LIN {X 0,Y 522.587,Z 549.53,A -85,B 0,C 180,E1 4793.93,E2 4793.93} C_VEL
LIN {X 0,Y 522.386,Z 549.53,A -85,B 0,C 180,E1 4799.594,E2 4799.594} C_VEL
LIN {X 0,Y 522.323,Z 549.53,A -85,B 0,C 180,E1 4805.74,E2 4805.74} C_VEL
LIN {X 0,Y 522.361,Z 549.53,A -85,B 0,C 180,E1 4811.419,E2 4811.419} C_VEL
LIN {X 0,Y 533.947,Z 582.684,A -85,B 0,C 180,E1 4813.515,E2 4813.515} C_VEL
LIN {X 0,Y 531.782,Z 621.229,A -85,B 0,C 180,E1 4815.534,E2 4815.534} C_VEL
LIN {X 0,Y 529.396,Z 657.061,A -85,B 0,C 180,E1 4818.174,E2 4818.174} C_VEL
LIN {X 0,Y 527.169,Z 689.396,A -85,B 0,C 180,E1 4821.377,E2 4821.377} C_VEL
LIN {X 0,Y 525.44,Z 717.104,A -85,B 0,C 180,E1 4824.999,E2 4824.999} C_VEL
LIN {X 0,Y 524.207,Z 740.402,A -85,B 0,C 180,E1 4829.059,E2 4829.059} C_VEL
LIN {X 0,Y 523.575,Z 757.4,A -85,B 0,C 180,E1 4833.13,E2 4833.13} C_VEL
LIN {X 0,Y 523.223,Z 768.491,A -85,B 0,C 180,E1 4837.003,E2 4837.003} C_VEL
LIN {X 0,Y 522.979,Z 775.702,A -85,B 0,C 180,E1 4841.427,E2 4841.427} C_VEL
LIN {X 0,Y 523.022,Z 777.495,A -85,B 0,C 180,E1 4844.895,E2 4844.895} C_VEL
LIN {X 0,Y 523.078,Z 775.878,A -85,B 0,C 180,E1 4848.307,E2 4848.307} C_VEL
LIN {X 0,Y 523.253,Z 769.377,A -85,B 0,C 180,E1 4852.515,E2 4852.515} C_VEL
LIN {X 0,Y 523.557,Z 757.742,A -85,B 0,C 180,E1 4856.681,E2 4856.681} C_VEL
LIN {X 0,Y 524.184,Z 739.509,A -85,B 0,C 180,E1 4861.031,E2 4861.031} C_VEL
LIN {X 0,Y 525.342,Z 716.823,A -85,B 0,C 180,E1 4864.956,E2 4864.956} C_VEL
LIN {X 0,Y 527.118,Z 690.017,A -85,B 0,C 180,E1 4868.461,E2 4868.461} C_VEL
LIN {X 0,Y 529.345,Z 658.044,A -85,B 0,C 180,E1 4871.65,E2 4871.65} C_VEL
LIN {X 0,Y 531.728,Z 622.755,A -85,B 0,C 180,E1 4874.276,E2 4874.276} C_VEL
LIN {X 0,Y 533.842,Z 585.818,A -85,B 0,C 180,E1 4876.253,E2 4876.253} C_VEL
LIN {X 0,Y 533.35,Z 577.741,A -85,B 0,C 180,E1 4876.653,E2 4876.653} C_VEL
LIN {X 0,Y 522.59,Z 549.53,A -85,B 0,C 180,E1 4878.475,E2 4878.475} C_VEL
LIN {X 0,Y 522.511,Z 549.53,A -85,B 0,C 180,E1 4879.609,E2 4879.609} C_VEL
LIN {X 0,Y 520.002,Z 549.53,A -85,B 0,C 180,E1 4881.019,E2 4881.019} C_VEL
LIN {X 0,Y 514.659,Z 549.53,A -85,B 0,C 180,E1 4883.132,E2 4883.132} C_VEL
LIN {X 0,Y 514.565,Z 549.53,A -85,B 0,C 180,E1 4883.376,E2 4883.376} C_VEL
LIN {X 0,Y 514.494,Z 549.53,A -85,B 0,C 180,E1 4888.085,E2 4888.085} C_VEL
LIN {X 0,Y 514.37,Z 549.53,A -85,B 0,C 180,E1 4894,E2 4894} C_VEL
LIN {X 0,Y 514.463,Z 549.53,A -85,B 0,C 180,E1 4900.344,E2 4900.344} C_VEL
LIN {X 0,Y 514.4,Z 549.53,A -85,B 0,C 180,E1 4905.056,E2 4905.056} C_VEL
LIN {X 0,Y 514.337,Z 549.53,A -85,B 0,C 180,E1 4911.816,E2 4911.816} C_VEL
LIN {X 0,Y 514.446,Z 549.53,A -85,B 0,C 180,E1 4914.365,E2 4914.365} C_VEL
LIN {X 0,Y 529.549,Z 582.461,A -85,B 0,C 180,E1 4916.004,E2 4916.004} C_VEL
LIN {X 0,Y 528.701,Z 628.433,A -85,B 0,C 180,E1 4916.908,E2 4916.908} C_VEL
LIN {X 0,Y 526.969,Z 666.113,A -85,B 0,C 180,E1 4918.265,E2 4918.265} C_VEL
LIN {X 0,Y 524.654,Z 702.724,A -85,B 0,C 180,E1 4920.246,E2 4920.246} C_VEL
LIN {X 0,Y 522.113,Z 737.095,A -85,B 0,C 180,E1 4922.823,E2 4922.823} C_VEL
LIN {X 0,Y 519.796,Z 768.223,A -85,B 0,C 180,E1 4925.933,E2 4925.933} C_VEL
LIN {X 0,Y 517.817,Z 795.232,A -85,B 0,C 180,E1 4929.459,E2 4929.459} C_VEL
LIN {X 0,Y 516.475,Z 818.065,A -85,B 0,C 180,E1 4933.391,E2 4933.391} C_VEL
LIN {X 0,Y 515.7,Z 834.826,A -85,B 0,C 180,E1 4937.279,E2 4937.279} C_VEL
LIN {X 0,Y 515.364,Z 847.612,A -85,B 0,C 180,E1 4941.552,E2 4941.552} C_VEL
LIN {X 0,Y 515.231,Z 853.932,A -85,B 0,C 180,E1 4944.942,E2 4944.942} C_VEL
LIN {X 0,Y 515.211,Z 857.084,A -85,B 0,C 180,E1 4948.315,E2 4948.315} C_VEL
LIN {X 0,Y 515.199,Z 856.636,A -85,B 0,C 180,E1 4952.428,E2 4952.428} C_VEL
LIN {X 0,Y 515.289,Z 851.182,A -85,B 0,C 180,E1 4956.749,E2 4956.749} C_VEL
LIN {X 0,Y 515.5,Z 841.923,A -85,B 0,C 180,E1 4960.589,E2 4960.589} C_VEL
LIN {X 0,Y 516.106,Z 826.652,A -85,B 0,C 180,E1 4964.776,E2 4964.776} C_VEL
LIN {X 0,Y 517.278,Z 804.95,A -85,B 0,C 180,E1 4969.003,E2 4969.003} C_VEL
LIN {X 0,Y 519.005,Z 778.608,A -85,B 0,C 180,E1 4972.821,E2 4972.821} C_VEL
LIN {X 0,Y 521.271,Z 748.093,A -85,B 0,C 180,E1 4976.175,E2 4976.175} C_VEL
LIN {X 0,Y 523.839,Z 713.836,A -85,B 0,C 180,E1 4979.007,E2 4979.007} C_VEL
LIN {X 0,Y 526.461,Z 675.681,A -85,B 0,C 180,E1 4981.288,E2 4981.288} C_VEL
LIN {X 0,Y 528.473,Z 635.637,A -85,B 0,C 180,E1 4982.884,E2 4982.884} C_VEL
LIN {X 0,Y 529.548,Z 593.899,A -85,B 0,C 180,E1 4983.813,E2 4983.813} C_VEL
LIN {X 0,Y 528.896,Z 580.557,A -85,B 0,C 180,E1 4984.075,E2 4984.075} C_VEL
LIN {X 0,Y 514.406,Z 549.53,A -85,B 0,C 180,E1 4985.73,E2 4985.73} C_VEL
LIN {X 0,Y 514.463,Z 549.53,A -85,B 0,C 180,E1 4990.349,E2 4990.349} C_VEL
LIN {X 0,Y 514.395,Z 549.53,A -85,B 0,C 180,E1 4995.063,E2 4995.063} C_VEL
LIN {X 0,Y 514.324,Z 549.53,A -85,B 0,C 180,E1 5001.821,E2 5001.821} C_VEL
LIN {X 0,Y 514.526,Z 549.53,A -85,B 0,C 180,E1 5008.022,E2 5008.022} C_VEL
LIN {X 0,Y 514.498,Z 549.53,A -85,B 0,C 180,E1 5013.81,E2 5013.81} C_VEL
LIN {X 0,Y 514.563,Z 549.53,A -85,B 0,C 180,E1 5019.328,E2 5019.328} C_VEL
LIN {X 0,Y 514.73,Z 549.53,A -85,B 0,C 180,E1 5024.653,E2 5024.653} C_VEL
LIN {X 0,Y 514.859,Z 549.53,A -85,B 0,C 180,E1 5029.841,E2 5029.841} C_VEL
LIN {X 0,Y 514.93,Z 549.53,A -85,B 0,C 180,E1 5034.943,E2 5034.943} C_VEL
LIN {X 0,Y 515.174,Z 549.53,A -85,B 0,C 180,E1 5041.688,E2 5041.688} C_VEL
LIN {X 0,Y 515.005,Z 549.53,A -85,B 0,C 180,E1 5046.757,E2 5046.757} C_VEL
LIN {X 0,Y 514.781,Z 549.53,A -85,B 0,C 180,E1 5051.884,E2 5051.884} C_VEL
LIN {X 0,Y 514.696,Z 549.53,A -85,B 0,C 180,E1 5057.111,E2 5057.111} C_VEL
LIN {X 0,Y 514.62,Z 549.53,A -85,B 0,C 180,E1 5062.49,E2 5062.49} C_VEL
LIN {X 0,Y 514.462,Z 549.53,A -85,B 0,C 180,E1 5068.095,E2 5068.095} C_VEL
LIN {X 0,Y 514.358,Z 549.53,A -85,B 0,C 180,E1 5074.01,E2 5074.01} C_VEL
LIN {X 0,Y 514.423,Z 549.53,A -85,B 0,C 180,E1 5080.358,E2 5080.358} C_VEL
LIN {X 0,Y 514.362,Z 549.53,A -85,B 0,C 180,E1 5085.054,E2 5085.054} C_VEL
LIN {X 0,Y 514.345,Z 549.53,A -85,B 0,C 180,E1 5089.942,E2 5089.942} C_VEL
LIN {X 0,Y 514.429,Z 549.53,A -85,B 0,C 180,E1 5096,E2 5096} C_VEL
LIN {X 0,Y 514.46,Z 549.53,A -85,B 0,C 180,E1 5101.999,E2 5101.999} C_VEL
LIN {X 0,Y 514.558,Z 549.53,A -85,B 0,C 180,E1 5107.511,E2 5107.511} C_VEL
LIN {X 0,Y 514.696,Z 549.53,A -85,B 0,C 180,E1 5112.893,E2 5112.893} C_VEL
LIN {X 0,Y 514.781,Z 549.53,A -85,B 0,C 180,E1 5118.12,E2 5118.12} C_VEL
LIN {X 0,Y 514.881,Z 549.53,A -85,B 0,C 180,E1 5123.246,E2 5123.246} C_VEL
LIN {X 0,Y 514.971,Z 549.53,A -85,B 0,C 180,E1 5128.524,E2 5128.524} C_VEL
LIN {X 0,Y 514.933,Z 549.53,A -85,B 0,C 180,E1 5133.372,E2 5133.372} C_VEL
LIN {X 0,Y 514.812,Z 549.53,A -85,B 0,C 180,E1 5138.457,E2 5138.457} C_VEL
LIN {X 0,Y 514.743,Z 549.53,A -85,B 0,C 180,E1 5143.904,E2 5143.904} C_VEL
LIN {X 0,Y 514.64,Z 549.53,A -85,B 0,C 180,E1 5149.7,E2 5149.7} C_VEL
LIN {X 0,Y 514.658,Z 549.53,A -85,B 0,C 180,E1 5154.323,E2 5154.323} C_VEL
LIN {X 0,Y 514.447,Z 549.53,A -85,B 0,C 180,E1 5160.022,E2 5160.022} C_VEL
LIN {X 0,Y 514.412,Z 549.53,A -85,B 0,C 180,E1 5166.063,E2 5166.063} C_VEL
LIN {X 0,Y 514.465,Z 550.037,A -85,B 0,C 180,E1 5170.866,E2 5170.866} C_VEL
LIN {X 0,Y 527.106,Z 583.478,A -85,B 0,C 180,E1 5173.098,E2 5173.098} C_VEL
LIN {X 0,Y 524.76,Z 621.631,A -85,B 0,C 180,E1 5175.128,E2 5175.128} C_VEL
LIN {X 0,Y 522.259,Z 655.644,A -85,B 0,C 180,E1 5177.647,E2 5177.647} C_VEL
LIN {X 0,Y 519.773,Z 688.501,A -85,B 0,C 180,E1 5180.915,E2 5180.915} C_VEL
LIN {X 0,Y 517.796,Z 716.835,A -85,B 0,C 180,E1 5184.65,E2 5184.65} C_VEL
LIN {X 0,Y 516.485,Z 739.169,A -85,B 0,C 180,E1 5188.564,E2 5188.564} C_VEL
LIN {X 0,Y 515.708,Z 757.505,A -85,B 0,C 180,E1 5192.977,E2 5192.977} C_VEL
LIN {X 0,Y 515.274,Z 769.934,A -85,B 0,C 180,E1 5197.54,E2 5197.54} C_VEL
LIN {X 0,Y 515.086,Z 775.461,A -85,B 0,C 180,E1 5201.132,E2 5201.132} C_VEL
LIN {X 0,Y 515.088,Z 777.462,A -85,B 0,C 180,E1 5204.657,E2 5204.657} C_VEL
LIN {X 0,Y 515.153,Z 776.109,A -85,B 0,C 180,E1 5208.124,E2 5208.124} C_VEL
LIN {X 0,Y 515.348,Z 769.867,A -85,B 0,C 180,E1 5212.399,E2 5212.399} C_VEL
LIN {X 0,Y 515.68,Z 758.507,A -85,B 0,C 180,E1 5216.63,E2 5216.63} C_VEL
LIN {X 0,Y 516.358,Z 740.653,A -85,B 0,C 180,E1 5221.047,E2 5221.047} C_VEL
LIN {X 0,Y 517.728,Z 716.827,A -85,B 0,C 180,E1 5225.263,E2 5225.263} C_VEL
LIN {X 0,Y 519.792,Z 688.415,A -85,B 0,C 180,E1 5229.004,E2 5229.004} C_VEL
LIN {X 0,Y 522.267,Z 655.937,A -85,B 0,C 180,E1 5232.235,E2 5232.235} C_VEL
LIN {X 0,Y 524.895,Z 620.24,A -85,B 0,C 180,E1 5234.87,E2 5234.87} C_VEL
LIN {X 0,Y 527.04,Z 581.921,A -85,B 0,C 180,E1 5236.891,E2 5236.891} C_VEL
LIN {X 0,Y 514.633,Z 549.53,A -85,B 0,C 180,E1 5239.082,E2 5239.082} C_VEL
LIN {X 0,Y 514.565,Z 549.53,A -85,B 0,C 180,E1 5243.376,E2 5243.376} C_VEL
LIN {X 0,Y 512.046,Z 549.53,A -85,B 0,C 180,E1 5244.81,E2 5244.81} C_VEL
LIN {X 0,Y 506.53,Z 549.53,A -85,B 0,C 180,E1 5247.208,E2 5247.208} C_VEL
LIN {X 0,Y 506.407,Z 549.53,A -85,B 0,C 180,E1 5253.158,E2 5253.158} C_VEL
LIN {X 0,Y 506.467,Z 549.53,A -85,B 0,C 180,E1 5258.988,E2 5258.988} C_VEL
LIN {X 0,Y 506.44,Z 549.53,A -85,B 0,C 180,E1 5264.15,E2 5264.15} C_VEL
LIN {X 0,Y 506.376,Z 549.53,A -85,B 0,C 180,E1 5268.867,E2 5268.867} C_VEL
LIN {X 0,Y 506.525,Z 549.563,A -85,B 0,C 180,E1 5273.887,E2 5273.887} C_VEL
LIN {X 0,Y 514.606,Z 567.373,A -85,B 0,C 180,E1 5274.676,E2 5274.676} C_VEL
LIN {X 0,Y 522.982,Z 584.842,A -85,B 0,C 180,E1 5275.556,E2 5275.556} C_VEL
LIN {X 0,Y 522.081,Z 628.432,A -85,B 0,C 180,E1 5276.433,E2 5276.433} C_VEL
LIN {X 0,Y 520.149,Z 666.955,A -85,B 0,C 180,E1 5277.842,E2 5277.842} C_VEL
LIN {X 0,Y 517.68,Z 702.721,A -85,B 0,C 180,E1 5279.804,E2 5279.804} C_VEL
LIN {X 0,Y 514.937,Z 737.092,A -85,B 0,C 180,E1 5282.412,E2 5282.412} C_VEL
LIN {X 0,Y 512.366,Z 768.222,A -85,B 0,C 180,E1 5285.561,E2 5285.561} C_VEL
LIN {X 0,Y 510.225,Z 795.231,A -85,B 0,C 180,E1 5289.139,E2 5289.139} C_VEL
LIN {X 0,Y 508.729,Z 818.063,A -85,B 0,C 180,E1 5293.131,E2 5293.131} C_VEL
LIN {X 0,Y 507.884,Z 834.827,A -85,B 0,C 180,E1 5297.08,E2 5297.08} C_VEL
LIN {X 0,Y 507.481,Z 847.612,A -85,B 0,C 180,E1 5301.42,E2 5301.42} C_VEL
LIN {X 0,Y 507.334,Z 853.932,A -85,B 0,C 180,E1 5304.863,E2 5304.863} C_VEL
LIN {X 0,Y 507.329,Z 857.084,A -85,B 0,C 180,E1 5308.289,E2 5308.289} C_VEL
LIN {X 0,Y 507.391,Z 857.086,A -85,B 0,C 180,E1 5311.709,E2 5311.709} C_VEL
LIN {X 0,Y 507.418,Z 852.726,A -85,B 0,C 180,E1 5315.994,E2 5315.994} C_VEL
LIN {X 0,Y 507.617,Z 843.214,A -85,B 0,C 180,E1 5320.309,E2 5320.309} C_VEL
LIN {X 0,Y 508.243,Z 827.853,A -85,B 0,C 180,E1 5324.727,E2 5324.727} C_VEL
LIN {X 0,Y 509.531,Z 806.274,A -85,B 0,C 180,E1 5329.078,E2 5329.078} C_VEL
LIN {X 0,Y 511.324,Z 781.087,A -85,B 0,C 180,E1 5332.858,E2 5332.858} C_VEL
LIN {X 0,Y 513.741,Z 751.547,A -85,B 0,C 180,E1 5336.235,E2 5336.235} C_VEL
LIN {X 0,Y 516.505,Z 717.528,A -85,B 0,C 180,E1 5339.169,E2 5339.169} C_VEL
LIN {X 0,Y 519.259,Z 681.482,A -85,B 0,C 180,E1 5341.44,E2 5341.44} C_VEL
LIN {X 0,Y 521.439,Z 645.004,A -85,B 0,C 180,E1 5343.038,E2 5343.038} C_VEL
LIN {X 0,Y 522.843,Z 606.759,A -85,B 0,C 180,E1 5344.069,E2 5344.069} C_VEL
LIN {X 0,Y 522.345,Z 583.286,A -85,B 0,C 180,E1 5344.517,E2 5344.517} C_VEL
LIN {X 0,Y 506.501,Z 549.53,A -85,B 0,C 180,E1 5346.278,E2 5346.278} C_VEL
LIN {X 0,Y 506.498,Z 549.53,A -85,B 0,C 180,E1 5351.648,E2 5351.648} C_VEL
LIN {X 0,Y 506.4,Z 549.53,A -85,B 0,C 180,E1 5356.561,E2 5356.561} C_VEL
LIN {X 0,Y 506.445,Z 549.53,A -85,B 0,C 180,E1 5363.285,E2 5363.285} C_VEL
LIN {X 0,Y 506.581,Z 549.53,A -85,B 0,C 180,E1 5369.468,E2 5369.468} C_VEL
LIN {X 0,Y 506.579,Z 549.53,A -85,B 0,C 180,E1 5375.269,E2 5375.269} C_VEL
LIN {X 0,Y 506.698,Z 549.53,A -85,B 0,C 180,E1 5380.815,E2 5380.815} C_VEL
LIN {X 0,Y 506.872,Z 549.53,A -85,B 0,C 180,E1 5386.179,E2 5386.179} C_VEL
LIN {X 0,Y 506.99,Z 549.53,A -85,B 0,C 180,E1 5391.416,E2 5391.416} C_VEL
LIN {X 0,Y 507.148,Z 549.53,A -85,B 0,C 180,E1 5396.581,E2 5396.581} C_VEL
LIN {X 0,Y 507.283,Z 549.53,A -85,B 0,C 180,E1 5401.714,E2 5401.714} C_VEL
LIN {X 0,Y 507.076,Z 549.53,A -85,B 0,C 180,E1 5406.863,E2 5406.863} C_VEL
LIN {X 0,Y 506.851,Z 549.53,A -85,B 0,C 180,E1 5412.073,E2 5412.073} C_VEL
LIN {X 0,Y 506.779,Z 549.53,A -85,B 0,C 180,E1 5417.387,E2 5417.387} C_VEL
LIN {X 0,Y 506.704,Z 549.53,A -85,B 0,C 180,E1 5422.861,E2 5422.861} C_VEL
LIN {X 0,Y 506.497,Z 549.53,A -85,B 0,C 180,E1 5428.577,E2 5428.577} C_VEL
LIN {X 0,Y 506.449,Z 549.53,A -85,B 0,C 180,E1 5434.615,E2 5434.615} C_VEL
LIN {X 0,Y 506.433,Z 549.53,A -85,B 0,C 180,E1 5441.13,E2 5441.13} C_VEL
LIN {X 0,Y 506.356,Z 549.53,A -85,B 0,C 180,E1 5446.551,E2 5446.551} C_VEL
LIN {X 0,Y 506.448,Z 549.53,A -85,B 0,C 180,E1 5453.28,E2 5453.28} C_VEL
LIN {X 0,Y 506.573,Z 549.53,A -85,B 0,C 180,E1 5459.463,E2 5459.463} C_VEL
LIN {X 0,Y 506.586,Z 549.53,A -85,B 0,C 180,E1 5465.266,E2 5465.266} C_VEL
LIN {X 0,Y 506.732,Z 549.53,A -85,B 0,C 180,E1 5470.813,E2 5470.813} C_VEL
LIN {X 0,Y 506.888,Z 549.53,A -85,B 0,C 180,E1 5476.176,E2 5476.176} C_VEL
LIN {X 0,Y 506.985,Z 549.53,A -85,B 0,C 180,E1 5481.413,E2 5481.413} C_VEL
LIN {X 0,Y 507.204,Z 549.53,A -85,B 0,C 180,E1 5486.578,E2 5486.578} C_VEL
LIN {X 0,Y 507.286,Z 549.53,A -85,B 0,C 180,E1 5491.711,E2 5491.711} C_VEL
LIN {X 0,Y 507.096,Z 549.53,A -85,B 0,C 180,E1 5496.86,E2 5496.86} C_VEL
LIN {X 0,Y 506.879,Z 549.53,A -85,B 0,C 180,E1 5502.07,E2 5502.07} C_VEL
LIN {X 0,Y 506.801,Z 549.53,A -85,B 0,C 180,E1 5507.383,E2 5507.383} C_VEL
LIN {X 0,Y 506.747,Z 549.53,A -85,B 0,C 180,E1 5512.857,E2 5512.857} C_VEL
LIN {X 0,Y 506.55,Z 549.53,A -85,B 0,C 180,E1 5518.571,E2 5518.571} C_VEL
LIN {X 0,Y 506.478,Z 549.53,A -85,B 0,C 180,E1 5524.611,E2 5524.611} C_VEL
LIN {X 0,Y 506.565,Z 549.913,A -85,B 0,C 180,E1 5530.288,E2 5530.288} C_VEL
LIN {X 0,Y 520.194,Z 586.345,A -85,B 0,C 180,E1 5532.764,E2 5532.764} C_VEL
LIN {X 0,Y 517.628,Z 624.022,A -85,B 0,C 180,E1 5534.842,E2 5534.842} C_VEL
LIN {X 0,Y 514.887,Z 657.943,A -85,B 0,C 180,E1 5537.439,E2 5537.439} C_VEL
LIN {X 0,Y 512.251,Z 689.781,A -85,B 0,C 180,E1 5540.693,E2 5540.693} C_VEL
LIN {X 0,Y 510.115,Z 717.806,A -85,B 0,C 180,E1 5544.485,E2 5544.485} C_VEL
LIN {X 0,Y 508.63,Z 740.964,A -85,B 0,C 180,E1 5548.676,E2 5548.676} C_VEL
LIN {X 0,Y 507.84,Z 758.04,A -85,B 0,C 180,E1 5552.954,E2 5552.954} C_VEL
LIN {X 0,Y 507.438,Z 769.407,A -85,B 0,C 180,E1 5557.174,E2 5557.174} C_VEL
LIN {X 0,Y 507.203,Z 775.22,A -85,B 0,C 180,E1 5560.827,E2 5560.827} C_VEL
LIN {X 0,Y 507.159,Z 777.428,A -85,B 0,C 180,E1 5564.411,E2 5564.411} C_VEL
LIN {X 0,Y 507.228,Z 776.315,A -85,B 0,C 180,E1 5567.936,E2 5567.936} C_VEL
LIN {X 0,Y 507.438,Z 770.348,A -85,B 0,C 180,E1 5572.28,E2 5572.28} C_VEL
LIN {X 0,Y 507.808,Z 759.271,A -85,B 0,C 180,E1 5576.578,E2 5576.578} C_VEL
LIN {X 0,Y 508.513,Z 742.718,A -85,B 0,C 180,E1 5580.849,E2 5580.849} C_VEL
LIN {X 0,Y 509.801,Z 721.169,A -85,B 0,C 180,E1 5584.894,E2 5584.894} C_VEL
LIN {X 0,Y 511.932,Z 693.978,A -85,B 0,C 180,E1 5588.714,E2 5588.714} C_VEL
LIN {X 0,Y 514.603,Z 662.054,A -85,B 0,C 180,E1 5592.097,E2 5592.097} C_VEL
LIN {X 0,Y 517.382,Z 627.987,A -85,B 0,C 180,E1 5594.801,E2 5594.801} C_VEL
LIN {X 0,Y 519.991,Z 590.057,A -85,B 0,C 180,E1 5596.975,E2 5596.975} C_VEL
LIN {X 0,Y 519.436,Z 582.65,A -85,B 0,C 180,E1 5597.381,E2 5597.381} C_VEL
LIN {X 0,Y 506.733,Z 549.53,A -85,B 0,C 180,E1 5599.669,E2 5599.669} C_VEL
LIN {X 0,Y 506.667,Z 549.53,A -85,B 0,C 180,E1 5604.726,E2 5604.726} C_VEL
LIN {X 0,Y 506.53,Z 549.53,A -85,B 0,C 180,E1 5607.208,E2 5607.208} C_VEL
LIN {X 0,Y 502.508,Z 549.53,A -85,B 0,C 180,E1 5609.137,E2 5609.137} C_VEL
LIN {X 0,Y 498.523,Z 549.53,A -85,B 0,C 180,E1 5611.097,E2 5611.097} C_VEL
LIN {X 0,Y 498.514,Z 549.53,A -85,B 0,C 180,E1 5617.398,E2 5617.398} C_VEL
LIN {X 0,Y 498.57,Z 549.53,A -85,B 0,C 180,E1 5623.21,E2 5623.21} C_VEL
LIN {X 0,Y 498.412,Z 549.53,A -85,B 0,C 180,E1 5629.408,E2 5629.408} C_VEL
LIN {X 0,Y 498.606,Z 549.912,A -85,B 0,C 180,E1 5633.373,E2 5633.373} C_VEL
LIN {X 0,Y 509.034,Z 572.438,A -85,B 0,C 180,E1 5634.412,E2 5634.412} C_VEL
LIN {X 0,Y 516.365,Z 586.575,A -85,B 0,C 180,E1 5635.085,E2 5635.085} C_VEL
LIN {X 0,Y 515.432,Z 629.878,A -85,B 0,C 180,E1 5635.988,E2 5635.988} C_VEL
LIN {X 0,Y 513.4,Z 666.952,A -85,B 0,C 180,E1 5637.367,E2 5637.367} C_VEL
LIN {X 0,Y 510.727,Z 702.986,A -85,B 0,C 180,E1 5639.368,E2 5639.368} C_VEL
LIN {X 0,Y 507.779,Z 737.089,A -85,B 0,C 180,E1 5641.989,E2 5641.989} C_VEL
LIN {X 0,Y 504.971,Z 768.222,A -85,B 0,C 180,E1 5645.179,E2 5645.179} C_VEL
LIN {X 0,Y 502.668,Z 795.229,A -85,B 0,C 180,E1 5648.81,E2 5648.81} C_VEL
LIN {X 0,Y 501,Z 818.062,A -85,B 0,C 180,E1 5652.862,E2 5652.862} C_VEL
LIN {X 0,Y 500.052,Z 834.828,A -85,B 0,C 180,E1 5656.874,E2 5656.874} C_VEL
LIN {X 0,Y 499.604,Z 847.612,A -85,B 0,C 180,E1 5661.284,E2 5661.284} C_VEL
LIN {X 0,Y 499.455,Z 853.932,A -85,B 0,C 180,E1 5664.781,E2 5664.781} C_VEL
LIN {X 0,Y 499.455,Z 857.084,A -85,B 0,C 180,E1 5668.262,E2 5668.262} C_VEL
LIN {X 0,Y 499.489,Z 857.086,A -85,B 0,C 180,E1 5671.736,E2 5671.736} C_VEL
LIN {X 0,Y 499.543,Z 852.726,A -85,B 0,C 180,E1 5676.089,E2 5676.089} C_VEL
LIN {X 0,Y 499.733,Z 843.214,A -85,B 0,C 180,E1 5680.473,E2 5680.473} C_VEL
LIN {X 0,Y 500.453,Z 827.498,A -85,B 0,C 180,E1 5685.051,E2 5685.051} C_VEL
LIN {X 0,Y 501.822,Z 806.273,A -85,B 0,C 180,E1 5689.382,E2 5689.382} C_VEL
LIN {X 0,Y 503.917,Z 780.07,A -85,B 0,C 180,E1 5693.349,E2 5693.349} C_VEL
LIN {X 0,Y 506.553,Z 750.393,A -85,B 0,C 180,E1 5696.756,E2 5696.756} C_VEL
LIN {X 0,Y 509.463,Z 717.576,A -85,B 0,C 180,E1 5699.608,E2 5699.608} C_VEL
LIN {X 0,Y 512.397,Z 681.751,A -85,B 0,C 180,E1 5701.894,E2 5701.894} C_VEL
LIN {X 0,Y 514.771,Z 645.205,A -85,B 0,C 180,E1 5703.514,E2 5703.514} C_VEL
LIN {X 0,Y 516.289,Z 607.121,A -85,B 0,C 180,E1 5704.555,E2 5704.555} C_VEL
LIN {X 0,Y 515.984,Z 586.327,A -85,B 0,C 180,E1 5704.946,E2 5704.946} C_VEL
LIN {X 0,Y 498.601,Z 549.53,A -85,B 0,C 180,E1 5706.865,E2 5706.865} C_VEL
LIN {X 0,Y 498.578,Z 549.53,A -85,B 0,C 180,E1 5713.219,E2 5713.219} C_VEL
LIN {X 0,Y 498.391,Z 549.53,A -85,B 0,C 180,E1 5719.417,E2 5719.417} C_VEL
LIN {X 0,Y 498.586,Z 549.53,A -85,B 0,C 180,E1 5725.075,E2 5725.075} C_VEL
LIN {X 0,Y 498.633,Z 549.53,A -85,B 0,C 180,E1 5730.938,E2 5730.938} C_VEL
LIN {X 0,Y 498.675,Z 549.53,A -85,B 0,C 180,E1 5736.757,E2 5736.757} C_VEL
LIN {X 0,Y 498.811,Z 549.53,A -85,B 0,C 180,E1 5742.334,E2 5742.334} C_VEL
LIN {X 0,Y 498.924,Z 549.53,A -85,B 0,C 180,E1 5747.74,E2 5747.74} C_VEL
LIN {X 0,Y 499.039,Z 549.53,A -85,B 0,C 180,E1 5753.033,E2 5753.033} C_VEL
LIN {X 0,Y 499.17,Z 549.53,A -85,B 0,C 180,E1 5758.266,E2 5758.266} C_VEL
LIN {X 0,Y 499.146,Z 549.53,A -85,B 0,C 180,E1 5763.482,E2 5763.482} C_VEL
LIN {X 0,Y 498.984,Z 549.53,A -85,B 0,C 180,E1 5768.73,E2 5768.73} C_VEL
LIN {X 0,Y 498.901,Z 549.53,A -85,B 0,C 180,E1 5774.054,E2 5774.054} C_VEL
LIN {X 0,Y 498.776,Z 549.53,A -85,B 0,C 180,E1 5779.778,E2 5779.778} C_VEL
LIN {X 0,Y 498.717,Z 549.53,A -85,B 0,C 180,E1 5785.156,E2 5785.156} C_VEL
LIN {X 0,Y 498.489,Z 549.53,A -85,B 0,C 180,E1 5791.741,E2 5791.741} C_VEL
LIN {X 0,Y 498.482,Z 549.53,A -85,B 0,C 180,E1 5797.843,E2 5797.843} C_VEL
LIN {X 0,Y 498.509,Z 549.53,A -85,B 0,C 180,E1 5804.315,E2 5804.315} C_VEL
LIN {X 0,Y 498.403,Z 549.53,A -85,B 0,C 180,E1 5810.362,E2 5810.362} C_VEL
LIN {X 0,Y 498.623,Z 549.53,A -85,B 0,C 180,E1 5816.869,E2 5816.869} C_VEL
LIN {X 0,Y 498.575,Z 549.53,A -85,B 0,C 180,E1 5822.903,E2 5822.903} C_VEL
LIN {X 0,Y 498.738,Z 549.53,A -85,B 0,C 180,E1 5828.637,E2 5828.637} C_VEL
LIN {X 0,Y 498.908,Z 549.53,A -85,B 0,C 180,E1 5834.15,E2 5834.15} C_VEL
LIN {X 0,Y 499.029,Z 549.53,A -85,B 0,C 180,E1 5839.512,E2 5839.512} C_VEL
LIN {X 0,Y 499.163,Z 549.53,A -85,B 0,C 180,E1 5844.78,E2 5844.78} C_VEL
LIN {X 0,Y 499.296,Z 549.53,A -85,B 0,C 180,E1 5850.001,E2 5850.001} C_VEL
LIN {X 0,Y 499.188,Z 549.53,A -85,B 0,C 180,E1 5855.221,E2 5855.221} C_VEL
LIN {X 0,Y 499.001,Z 549.53,A -85,B 0,C 180,E1 5860.49,E2 5860.49} C_VEL
LIN {X 0,Y 498.91,Z 549.53,A -85,B 0,C 180,E1 5865.851,E2 5865.851} C_VEL
LIN {X 0,Y 498.826,Z 549.53,A -85,B 0,C 180,E1 5871.361,E2 5871.361} C_VEL
LIN {X 0,Y 498.675,Z 549.53,A -85,B 0,C 180,E1 5877.093,E2 5877.093} C_VEL
LIN {X 0,Y 498.542,Z 549.53,A -85,B 0,C 180,E1 5883.139,E2 5883.139} C_VEL
LIN {X 0,Y 498.606,Z 549.53,A -85,B 0,C 180,E1 5889.667,E2 5889.667} C_VEL
LIN {X 0,Y 513.306,Z 588.442,A -85,B 0,C 180,E1 5892.384,E2 5892.384} C_VEL
LIN {X 0,Y 510.528,Z 626.132,A -85,B 0,C 180,E1 5894.53,E2 5894.53} C_VEL
LIN {X 0,Y 507.454,Z 660.876,A -85,B 0,C 180,E1 5897.284,E2 5897.284} C_VEL
LIN {X 0,Y 504.658,Z 692.14,A -85,B 0,C 180,E1 5900.595,E2 5900.595} C_VEL
LIN {X 0,Y 502.351,Z 719.717,A -85,B 0,C 180,E1 5904.467,E2 5904.467} C_VEL
LIN {X 0,Y 500.753,Z 742.446,A -85,B 0,C 180,E1 5908.746,E2 5908.746} C_VEL
LIN {X 0,Y 499.949,Z 758.736,A -85,B 0,C 180,E1 5912.979,E2 5912.979} C_VEL
LIN {X 0,Y 499.512,Z 770.127,A -85,B 0,C 180,E1 5917.399,E2 5917.399} C_VEL
LIN {X 0,Y 499.303,Z 774.958,A -85,B 0,C 180,E1 5920.512,E2 5920.512} C_VEL
LIN {X 0,Y 499.24,Z 777.386,A -85,B 0,C 180,E1 5924.157,E2 5924.157} C_VEL
LIN {X 0,Y 499.304,Z 776.479,A -85,B 0,C 180,E1 5927.742,E2 5927.742} C_VEL
LIN {X 0,Y 499.546,Z 770.776,A -85,B 0,C 180,E1 5932.158,E2 5932.158} C_VEL
LIN {X 0,Y 499.938,Z 760.008,A -85,B 0,C 180,E1 5936.524,E2 5936.524} C_VEL
LIN {X 0,Y 500.673,Z 743.784,A -85,B 0,C 180,E1 5940.863,E2 5940.863} C_VEL
LIN {X 0,Y 502.142,Z 721.323,A -85,B 0,C 180,E1 5945.186,E2 5945.186} C_VEL
LIN {X 0,Y 504.475,Z 694.176,A -85,B 0,C 180,E1 5949.062,E2 5949.062} C_VEL
LIN {X 0,Y 507.356,Z 662.322,A -85,B 0,C 180,E1 5952.491,E2 5952.491} C_VEL
LIN {X 0,Y 510.472,Z 626.987,A -85,B 0,C 180,E1 5955.321,E2 5955.321} C_VEL
LIN {X 0,Y 513.206,Z 590.675,A -85,B 0,C 180,E1 5957.418,E2 5957.418} C_VEL
LIN {X 0,Y 512.018,Z 583.901,A -85,B 0,C 180,E1 5957.847,E2 5957.847} C_VEL
LIN {X 0,Y 498.808,Z 549.53,A -85,B 0,C 180,E1 5960.192,E2 5960.192} C_VEL
LIN {X 0,Y 498.744,Z 549.53,A -85,B 0,C 180,E1 5965.146,E2 5965.146} C_VEL
LIN {X 0,Y 498.523,Z 549.53,A -85,B 0,C 180,E1 5971.097,E2 5971.097} C_VEL
LIN {X 0,Y 497.218,Z 549.53,A -85,B 0,C 180,E1 5972.094,E2 5972.094} C_VEL
LIN {X 0,Y 490.579,Z 549.53,A -85,B 0,C 180,E1 5974.811,E2 5974.811} C_VEL
LIN {X 0,Y 490.492,Z 549.53,A -85,B 0,C 180,E1 5975.069,E2 5975.069} C_VEL
LIN {X 0,Y 490.597,Z 549.53,A -85,B 0,C 180,E1 5980.392,E2 5980.392} C_VEL
LIN {X 0,Y 490.606,Z 549.53,A -85,B 0,C 180,E1 5985.212,E2 5985.212} C_VEL
LIN {X 0,Y 490.52,Z 549.53,A -85,B 0,C 180,E1 5991.878,E2 5991.878} C_VEL
LIN {X 0,Y 490.606,Z 549.53,A -85,B 0,C 180,E1 5992.793,E2 5992.793} C_VEL
LIN {X 0,Y 502.905,Z 576.614,A -85,B 0,C 180,E1 5994.092,E2 5994.092} C_VEL
LIN {X 0,Y 509.549,Z 589.623,A -85,B 0,C 180,E1 5994.713,E2 5994.713} C_VEL
LIN {X 0,Y 508.506,Z 633.83,A -85,B 0,C 180,E1 5995.648,E2 5995.648} C_VEL
LIN {X 0,Y 506.446,Z 670.712,A -85,B 0,C 180,E1 5997.059,E2 5997.059} C_VEL
LIN {X 0,Y 503.378,Z 708.075,A -85,B 0,C 180,E1 5999.247,E2 5999.247} C_VEL
LIN {X 0,Y 499.985,Z 743.846,A -85,B 0,C 180,E1 6002.172,E2 6002.172} C_VEL
LIN {X 0,Y 496.857,Z 776.091,A -85,B 0,C 180,E1 6005.757,E2 6005.757} C_VEL
LIN {X 0,Y 494.434,Z 802.171,A -85,B 0,C 180,E1 6009.594,E2 6009.594} C_VEL
LIN {X 0,Y 492.901,Z 822.299,A -85,B 0,C 180,E1 6013.492,E2 6013.492} C_VEL
LIN {X 0,Y 492.014,Z 837.895,A -85,B 0,C 180,E1 6017.56,E2 6017.56} C_VEL
LIN {X 0,Y 491.679,Z 849.535,A -85,B 0,C 180,E1 6022.034,E2 6022.034} C_VEL
LIN {X 0,Y 491.491,Z 855.896,A -85,B 0,C 180,E1 6026.467,E2 6026.467} C_VEL
LIN {X 0,Y 491.539,Z 857.5,A -85,B 0,C 180,E1 6029.999,E2 6029.999} C_VEL
LIN {X 0,Y 491.497,Z 855.9,A -85,B 0,C 180,E1 6033.531,E2 6033.531} C_VEL
LIN {X 0,Y 491.697,Z 849.541,A -85,B 0,C 180,E1 6037.964,E2 6037.964} C_VEL
LIN {X 0,Y 492.109,Z 837.903,A -85,B 0,C 180,E1 6042.436,E2 6042.436} C_VEL
LIN {X 0,Y 493.152,Z 820.237,A -85,B 0,C 180,E1 6046.957,E2 6046.957} C_VEL
LIN {X 0,Y 494.829,Z 797.841,A -85,B 0,C 180,E1 6051.121,E2 6051.121} C_VEL
LIN {X 0,Y 497.289,Z 771.449,A -85,B 0,C 180,E1 6054.826,E2 6054.826} C_VEL
LIN {X 0,Y 500.363,Z 740.195,A -85,B 0,C 180,E1 6058.161,E2 6058.161} C_VEL
LIN {X 0,Y 503.551,Z 706.243,A -85,B 0,C 180,E1 6060.876,E2 6060.876} C_VEL
LIN {X 0,Y 506.468,Z 669.667,A -85,B 0,C 180,E1 6062.994,E2 6062.994} C_VEL
LIN {X 0,Y 508.676,Z 631.394,A -85,B 0,C 180,E1 6064.438,E2 6064.438} C_VEL
LIN {X 0,Y 509.281,Z 588.801,A -85,B 0,C 180,E1 6065.386,E2 6065.386} C_VEL
LIN {X 0,Y 490.619,Z 549.53,A -85,B 0,C 180,E1 6067.549,E2 6067.549} C_VEL
LIN {X 0,Y 490.669,Z 549.53,A -85,B 0,C 180,E1 6072.753,E2 6072.753} C_VEL
LIN {X 0,Y 490.54,Z 549.53,A -85,B 0,C 180,E1 6077.796,E2 6077.796} C_VEL
LIN {X 0,Y 490.555,Z 549.53,A -85,B 0,C 180,E1 6084.102,E2 6084.102} C_VEL
LIN {X 0,Y 490.668,Z 549.53,A -85,B 0,C 180,E1 6090.42,E2 6090.42} C_VEL
LIN {X 0,Y 490.751,Z 549.53,A -85,B 0,C 180,E1 6096.359,E2 6096.359} C_VEL
LIN {X 0,Y 490.904,Z 549.53,A -85,B 0,C 180,E1 6102.96,E2 6102.96} C_VEL
LIN {X 0,Y 491.085,Z 549.53,A -85,B 0,C 180,E1 6109.344,E2 6109.344} C_VEL
LIN {X 0,Y 491.21,Z 549.53,A -85,B 0,C 180,E1 6114.698,E2 6114.698} C_VEL
LIN {X 0,Y 491.339,Z 549.53,A -85,B 0,C 180,E1 6120.004,E2 6120.004} C_VEL
LIN {X 0,Y 491.259,Z 549.53,A -85,B 0,C 180,E1 6125.309,E2 6125.309} C_VEL
LIN {X 0,Y 491.068,Z 549.53,A -85,B 0,C 180,E1 6130.664,E2 6130.664} C_VEL
LIN {X 0,Y 490.926,Z 549.53,A -85,B 0,C 180,E1 6137.048,E2 6137.048} C_VEL
LIN {X 0,Y 490.816,Z 549.53,A -85,B 0,C 180,E1 6143.645,E2 6143.645} C_VEL
LIN {X 0,Y 490.593,Z 549.53,A -85,B 0,C 180,E1 6150.218,E2 6150.218} C_VEL
LIN {X 0,Y 490.531,Z 549.53,A -85,B 0,C 180,E1 6156.631,E2 6156.631} C_VEL
LIN {X 0,Y 490.601,Z 549.53,A -85,B 0,C 180,E1 6162.765,E2 6162.765} C_VEL
LIN {X 0,Y 490.508,Z 549.53,A -85,B 0,C 180,E1 6167.805,E2 6167.805} C_VEL
LIN {X 0,Y 490.548,Z 549.53,A -85,B 0,C 180,E1 6174.097,E2 6174.097} C_VEL
LIN {X 0,Y 490.642,Z 549.53,A -85,B 0,C 180,E1 6180.414,E2 6180.414} C_VEL
LIN {X 0,Y 490.752,Z 549.53,A -85,B 0,C 180,E1 6186.355,E2 6186.355} C_VEL
LIN {X 0,Y 490.937,Z 549.53,A -85,B 0,C 180,E1 6192.958,E2 6192.958} C_VEL
LIN {X 0,Y 491.111,Z 549.53,A -85,B 0,C 180,E1 6199.341,E2 6199.341} C_VEL
LIN {X 0,Y 491.246,Z 549.53,A -85,B 0,C 180,E1 6204.695,E2 6204.695} C_VEL
LIN {X 0,Y 491.395,Z 549.53,A -85,B 0,C 180,E1 6210.001,E2 6210.001} C_VEL
LIN {X 0,Y 491.276,Z 549.53,A -85,B 0,C 180,E1 6215.306,E2 6215.306} C_VEL
LIN {X 0,Y 491.09,Z 549.53,A -85,B 0,C 180,E1 6220.661,E2 6220.661} C_VEL
LIN {X 0,Y 490.946,Z 549.53,A -85,B 0,C 180,E1 6227.046,E2 6227.046} C_VEL
LIN {X 0,Y 490.866,Z 549.53,A -85,B 0,C 180,E1 6233.64,E2 6233.64} C_VEL
LIN {X 0,Y 490.629,Z 549.53,A -85,B 0,C 180,E1 6240.219,E2 6240.219} C_VEL
LIN {X 0,Y 490.571,Z 549.53,A -85,B 0,C 180,E1 6245.903,E2 6245.903} C_VEL
LIN {X 0,Y 490.61,Z 549.638,A -85,B 0,C 180,E1 6249.063,E2 6249.063} C_VEL
LIN {X 0,Y 505.648,Z 588.827,A -85,B 0,C 180,E1 6251.851,E2 6251.851} C_VEL
LIN {X 0,Y 505.783,Z 599.641,A -85,B 0,C 180,E1 6252.462,E2 6252.462} C_VEL
LIN {X 0,Y 502.7,Z 635.866,A -85,B 0,C 180,E1 6254.762,E2 6254.762} C_VEL
LIN {X 0,Y 499.384,Z 670.324,A -85,B 0,C 180,E1 6257.767,E2 6257.767} C_VEL
LIN {X 0,Y 496.35,Z 701.154,A -85,B 0,C 180,E1 6261.374,E2 6261.374} C_VEL
LIN {X 0,Y 494.039,Z 727.059,A -85,B 0,C 180,E1 6265.393,E2 6265.393} C_VEL
LIN {X 0,Y 492.653,Z 747.448,A -85,B 0,C 180,E1 6269.654,E2 6269.654} C_VEL
LIN {X 0,Y 491.884,Z 761.846,A -85,B 0,C 180,E1 6273.821,E2 6273.821} C_VEL
LIN {X 0,Y 491.549,Z 771.952,A -85,B 0,C 180,E1 6278.304,E2 6278.304} C_VEL
LIN {X 0,Y 491.3,Z 776.909,A -85,B 0,C 180,E1 6282.815,E2 6282.815} C_VEL
LIN {X 0,Y 491.401,Z 776.642,A -85,B 0,C 180,E1 6287.541,E2 6287.541} C_VEL
LIN {X 0,Y 491.64,Z 771.204,A -85,B 0,C 180,E1 6292.031,E2 6292.031} C_VEL
LIN {X 0,Y 492.058,Z 760.739,A -85,B 0,C 180,E1 6296.468,E2 6296.468} C_VEL
LIN {X 0,Y 492.847,Z 744.844,A -85,B 0,C 180,E1 6300.876,E2 6300.876} C_VEL
LIN {X 0,Y 494.402,Z 722.753,A -85,B 0,C 180,E1 6305.268,E2 6305.268} C_VEL
LIN {X 0,Y 496.862,Z 696.086,A -85,B 0,C 180,E1 6309.202,E2 6309.202} C_VEL
LIN {X 0,Y 499.989,Z 664.875,A -85,B 0,C 180,E1 6312.678,E2 6312.678} C_VEL
LIN {X 0,Y 503.308,Z 629.875,A -85,B 0,C 180,E1 6315.58,E2 6315.58} C_VEL
LIN {X 0,Y 506.357,Z 592.327,A -85,B 0,C 180,E1 6317.82,E2 6317.82} C_VEL
LIN {X 0,Y 497.983,Z 568.076,A -85,B 0,C 180,E1 6319.534,E2 6319.534} C_VEL
LIN {X 0,Y 490.916,Z 549.53,A -85,B 0,C 180,E1 6320.778,E2 6320.778} C_VEL
LIN {X 0,Y 490.715,Z 549.53,A -85,B 0,C 180,E1 6326.519,E2 6326.519} C_VEL
LIN {X 0,Y 490.641,Z 549.53,A -85,B 0,C 180,E1 6331.636,E2 6331.636} C_VEL
LIN {X 0,Y 490.492,Z 549.53,A -85,B 0,C 180,E1 6335.069,E2 6335.069} C_VEL
LIN {X 0,Y 488.053,Z 549.53,A -85,B 0,C 180,E1 6336.573,E2 6336.573} C_VEL
LIN {X 0,Y 482.62,Z 549.53,A -85,B 0,C 180,E1 6339.09,E2 6339.09} C_VEL
LIN {X 0,Y 482.661,Z 549.53,A -85,B 0,C 180,E1 6343.821,E2 6343.821} C_VEL
LIN {X 0,Y 482.565,Z 549.53,A -85,B 0,C 180,E1 6348.844,E2 6348.844} C_VEL
LIN {X 0,Y 482.684,Z 550.102,A -85,B 0,C 180,E1 6352.271,E2 6352.271} C_VEL
LIN {X 0,Y 498.869,Z 584.539,A -85,B 0,C 180,E1 6353.96,E2 6353.96} C_VEL
LIN {X 0,Y 502.649,Z 592.509,A -85,B 0,C 180,E1 6354.329,E2 6354.329} C_VEL
LIN {X 0,Y 501.308,Z 636.476,A -85,B 0,C 180,E1 6355.322,E2 6355.322} C_VEL
LIN {X 0,Y 498.979,Z 677.092,A -85,B 0,C 180,E1 6356.959,E2 6356.959} C_VEL
LIN {X 0,Y 496.21,Z 711.412,A -85,B 0,C 180,E1 6359.008,E2 6359.008} C_VEL
LIN {X 0,Y 492.616,Z 745.768,A -85,B 0,C 180,E1 6361.924,E2 6361.924} C_VEL
LIN {X 0,Y 489.376,Z 776.592,A -85,B 0,C 180,E1 6365.432,E2 6365.432} C_VEL
LIN {X 0,Y 486.762,Z 802.942,A -85,B 0,C 180,E1 6369.397,E2 6369.397} C_VEL
LIN {X 0,Y 485.192,Z 822.299,A -85,B 0,C 180,E1 6373.222,E2 6373.222} C_VEL
LIN {X 0,Y 484.116,Z 839.278,A -85,B 0,C 180,E1 6377.812,E2 6377.812} C_VEL
LIN {X 0,Y 483.803,Z 849.535,A -85,B 0,C 180,E1 6381.903,E2 6381.903} C_VEL
LIN {X 0,Y 483.593,Z 855.896,A -85,B 0,C 180,E1 6386.409,E2 6386.409} C_VEL
LIN {X 0,Y 483.654,Z 857.5,A -85,B 0,C 180,E1 6389.999,E2 6389.999} C_VEL
LIN {X 0,Y 483.602,Z 855.9,A -85,B 0,C 180,E1 6393.589,E2 6393.589} C_VEL
LIN {X 0,Y 483.827,Z 849.541,A -85,B 0,C 180,E1 6398.095,E2 6398.095} C_VEL
LIN {X 0,Y 484.282,Z 837.902,A -85,B 0,C 180,E1 6402.641,E2 6402.641} C_VEL
LIN {X 0,Y 485.355,Z 820.262,A -85,B 0,C 180,E1 6407.232,E2 6407.232} C_VEL
LIN {X 0,Y 487.287,Z 797.911,A -85,B 0,C 180,E1 6411.452,E2 6411.452} C_VEL
LIN {X 0,Y 489.981,Z 771.084,A -85,B 0,C 180,E1 6415.268,E2 6415.268} C_VEL
LIN {X 0,Y 493.229,Z 740.61,A -85,B 0,C 180,E1 6418.564,E2 6418.564} C_VEL
LIN {X 0,Y 496.495,Z 708.084,A -85,B 0,C 180,E1 6421.225,E2 6421.225} C_VEL
LIN {X 0,Y 499.469,Z 670.414,A -85,B 0,C 180,E1 6423.404,E2 6423.404} C_VEL
LIN {X 0,Y 501.94,Z 630.612,A -85,B 0,C 180,E1 6424.924,E2 6424.924} C_VEL
LIN {X 0,Y 502.634,Z 591.492,A -85,B 0,C 180,E1 6425.82,E2 6425.82} C_VEL
LIN {X 0,Y 482.696,Z 549.53,A -85,B 0,C 180,E1 6428.184,E2 6428.184} C_VEL
LIN {X 0,Y 482.663,Z 549.53,A -85,B 0,C 180,E1 6433.83,E2 6433.83} C_VEL
LIN {X 0,Y 482.554,Z 549.53,A -85,B 0,C 180,E1 6438.852,E2 6438.852} C_VEL
LIN {X 0,Y 482.622,Z 549.53,A -85,B 0,C 180,E1 6444.652,E2 6444.652} C_VEL
LIN {X 0,Y 482.776,Z 549.53,A -85,B 0,C 180,E1 6449.887,E2 6449.887} C_VEL
LIN {X 0,Y 482.795,Z 549.53,A -85,B 0,C 180,E1 6455.945,E2 6455.945} C_VEL
LIN {X 0,Y 482.946,Z 549.53,A -85,B 0,C 180,E1 6461.734,E2 6461.734} C_VEL
LIN {X 0,Y 483.092,Z 549.53,A -85,B 0,C 180,E1 6467.331,E2 6467.331} C_VEL
LIN {X 0,Y 483.229,Z 549.53,A -85,B 0,C 180,E1 6472.804,E2 6472.804} C_VEL
LIN {X 0,Y 483.383,Z 549.53,A -85,B 0,C 180,E1 6478.209,E2 6478.209} C_VEL
LIN {X 0,Y 483.34,Z 549.53,A -85,B 0,C 180,E1 6483.596,E2 6483.596} C_VEL
LIN {X 0,Y 483.16,Z 549.53,A -85,B 0,C 180,E1 6489.018,E2 6489.018} C_VEL
LIN {X 0,Y 483.057,Z 549.53,A -85,B 0,C 180,E1 6494.525,E2 6494.525} C_VEL
LIN {X 0,Y 482.955,Z 549.53,A -85,B 0,C 180,E1 6500.176,E2 6500.176} C_VEL
LIN {X 0,Y 482.836,Z 549.53,A -85,B 0,C 180,E1 6506.044,E2 6506.044} C_VEL
LIN {X 0,Y 482.654,Z 549.53,A -85,B 0,C 180,E1 6512.231,E2 6512.231} C_VEL
LIN {X 0,Y 482.631,Z 549.53,A -85,B 0,C 180,E1 6518.864,E2 6518.864} C_VEL
LIN {X 0,Y 482.617,Z 549.53,A -85,B 0,C 180,E1 6523.818,E2 6523.818} C_VEL
LIN {X 0,Y 482.536,Z 549.53,A -85,B 0,C 180,E1 6528.86,E2 6528.86} C_VEL
LIN {X 0,Y 482.623,Z 549.53,A -85,B 0,C 180,E1 6534.657,E2 6534.657} C_VEL
LIN {X 0,Y 482.745,Z 549.53,A -85,B 0,C 180,E1 6539.88,E2 6539.88} C_VEL
LIN {X 0,Y 482.793,Z 549.53,A -85,B 0,C 180,E1 6545.941,E2 6545.941} C_VEL
LIN {X 0,Y 482.979,Z 549.53,A -85,B 0,C 180,E1 6551.731,E2 6551.731} C_VEL
LIN {X 0,Y 483.111,Z 549.53,A -85,B 0,C 180,E1 6557.328,E2 6557.328} C_VEL
LIN {X 0,Y 483.247,Z 549.53,A -85,B 0,C 180,E1 6562.801,E2 6562.801} C_VEL
LIN {X 0,Y 483.412,Z 549.53,A -85,B 0,C 180,E1 6568.206,E2 6568.206} C_VEL
LIN {X 0,Y 483.333,Z 549.53,A -85,B 0,C 180,E1 6573.593,E2 6573.593} C_VEL
LIN {X 0,Y 483.179,Z 549.53,A -85,B 0,C 180,E1 6579.015,E2 6579.015} C_VEL
LIN {X 0,Y 483.085,Z 549.53,A -85,B 0,C 180,E1 6584.522,E2 6584.522} C_VEL
LIN {X 0,Y 482.979,Z 549.53,A -85,B 0,C 180,E1 6590.172,E2 6590.172} C_VEL
LIN {X 0,Y 482.888,Z 549.53,A -85,B 0,C 180,E1 6596.039,E2 6596.039} C_VEL
LIN {X 0,Y 482.702,Z 549.53,A -85,B 0,C 180,E1 6602.225,E2 6602.225} C_VEL
LIN {X 0,Y 482.683,Z 549.836,A -85,B 0,C 180,E1 6608.429,E2 6608.429} C_VEL
LIN {X 0,Y 497.77,Z 588.565,A -85,B 0,C 180,E1 6611.271,E2 6611.271} C_VEL
LIN {X 0,Y 499.27,Z 596.624,A -85,B 0,C 180,E1 6611.821,E2 6611.821} C_VEL
LIN {X 0,Y 496.044,Z 632.996,A -85,B 0,C 180,E1 6614.079,E2 6614.079} C_VEL
LIN {X 0,Y 492.487,Z 667.306,A -85,B 0,C 180,E1 6617.033,E2 6617.033} C_VEL
LIN {X 0,Y 489.316,Z 697.506,A -85,B 0,C 180,E1 6620.5,E2 6620.5} C_VEL
LIN {X 0,Y 486.684,Z 724.404,A -85,B 0,C 180,E1 6624.604,E2 6624.604} C_VEL
LIN {X 0,Y 484.951,Z 746.314,A -85,B 0,C 180,E1 6629.119,E2 6629.119} C_VEL
LIN {X 0,Y 484.115,Z 761.078,A -85,B 0,C 180,E1 6633.368,E2 6633.368} C_VEL
LIN {X 0,Y 483.669,Z 771.5,A -85,B 0,C 180,E1 6637.932,E2 6637.932} C_VEL
LIN {X 0,Y 483.421,Z 776.259,A -85,B 0,C 180,E1 6641.744,E2 6641.744} C_VEL
LIN {X 0,Y 483.431,Z 777.322,A -85,B 0,C 180,E1 6646.146,E2 6646.146} C_VEL
LIN {X 0,Y 483.711,Z 773.073,A -85,B 0,C 180,E1 6650.992,E2 6650.992} C_VEL
LIN {X 0,Y 484.08,Z 763.892,A -85,B 0,C 180,E1 6655.512,E2 6655.512} C_VEL
LIN {X 0,Y 484.824,Z 749.46,A -85,B 0,C 180,E1 6659.996,E2 6659.996} C_VEL
LIN {X 0,Y 486.176,Z 729.584,A -85,B 0,C 180,E1 6664.362,E2 6664.362} C_VEL
LIN {X 0,Y 488.641,Z 704.455,A -85,B 0,C 180,E1 6668.46,E2 6668.46} C_VEL
LIN {X 0,Y 491.801,Z 673.759,A -85,B 0,C 180,E1 6672.215,E2 6672.215} C_VEL
LIN {X 0,Y 495.341,Z 640.055,A -85,B 0,C 180,E1 6675.293,E2 6675.293} C_VEL
LIN {X 0,Y 498.597,Z 604.212,A -85,B 0,C 180,E1 6677.674,E2 6677.674} C_VEL
LIN {X 0,Y 498.831,Z 591.023,A -85,B 0,C 180,E1 6678.407,E2 6678.407} C_VEL
LIN {X 0,Y 484.811,Z 555.132,A -85,B 0,C 180,E1 6680.961,E2 6680.961} C_VEL
LIN {X 0,Y 482.994,Z 549.53,A -85,B 0,C 180,E1 6681.387,E2 6681.387} C_VEL
LIN {X 0,Y 482.856,Z 549.53,A -85,B 0,C 180,E1 6686.035,E2 6686.035} C_VEL
LIN {X 0,Y 482.697,Z 549.53,A -85,B 0,C 180,E1 6692.219,E2 6692.219} C_VEL
LIN {X 0,Y 482.655,Z 549.53,A -85,B 0,C 180,E1 6698.852,E2 6698.852} C_VEL
LIN {X 0,Y 482.62,Z 549.53,A -85,B 0,C 180,E1 6699.09,E2 6699.09} C_VEL
LIN {X 0,Y 478.61,Z 549.53,A -85,B 0,C 180,E1 6701.114,E2 6701.114} C_VEL
LIN {X 0,Y 474.633,Z 549.53,A -85,B 0,C 180,E1 6703.171,E2 6703.171} C_VEL
LIN {X 0,Y 474.583,Z 549.53,A -85,B 0,C 180,E1 6707.935,E2 6707.935} C_VEL
LIN {X 0,Y 474.723,Z 549.555,A -85,B 0,C 180,E1 6711.662,E2 6711.662} C_VEL
LIN {X 0,Y 492.331,Z 587.906,A -85,B 0,C 180,E1 6713.586,E2 6713.586} C_VEL
LIN {X 0,Y 495.668,Z 594.335,A -85,B 0,C 180,E1 6713.911,E2 6713.911} C_VEL
LIN {X 0,Y 494.21,Z 637.114,A -85,B 0,C 180,E1 6714.932,E2 6714.932} C_VEL
LIN {X 0,Y 491.783,Z 676.369,A -85,B 0,C 180,E1 6716.544,E2 6716.544} C_VEL
LIN {X 0,Y 488.774,Z 713.562,A -85,B 0,C 180,E1 6718.78,E2 6718.78} C_VEL
LIN {X 0,Y 485.659,Z 744.511,A -85,B 0,C 180,E1 6721.347,E2 6721.347} C_VEL
LIN {X 0,Y 482.119,Z 775.733,A -85,B 0,C 180,E1 6724.915,E2 6724.915} C_VEL
LIN {X 0,Y 479.259,Z 801.995,A -85,B 0,C 180,E1 6728.886,E2 6728.886} C_VEL
LIN {X 0,Y 477.435,Z 822.632,A -85,B 0,C 180,E1 6733.021,E2 6733.021} C_VEL
LIN {X 0,Y 476.259,Z 839.279,A -85,B 0,C 180,E1 6737.608,E2 6737.608} C_VEL
LIN {X 0,Y 475.932,Z 849.535,A -85,B 0,C 180,E1 6741.769,E2 6741.769} C_VEL
LIN {X 0,Y 475.689,Z 855.896,A -85,B 0,C 180,E1 6746.349,E2 6746.349} C_VEL
LIN {X 0,Y 475.754,Z 857.5,A -85,B 0,C 180,E1 6749.999,E2 6749.999} C_VEL
LIN {X 0,Y 475.7,Z 855.9,A -85,B 0,C 180,E1 6753.649,E2 6753.649} C_VEL
LIN {X 0,Y 475.959,Z 849.541,A -85,B 0,C 180,E1 6758.229,E2 6758.229} C_VEL
LIN {X 0,Y 476.458,Z 837.902,A -85,B 0,C 180,E1 6762.852,E2 6762.852} C_VEL
LIN {X 0,Y 477.583,Z 821.011,A -85,B 0,C 180,E1 6767.357,E2 6767.357} C_VEL
LIN {X 0,Y 479.71,Z 797.907,A -85,B 0,C 180,E1 6771.808,E2 6771.808} C_VEL
LIN {X 0,Y 482.72,Z 770.343,A -85,B 0,C 180,E1 6775.772,E2 6775.772} C_VEL
LIN {X 0,Y 486.149,Z 740.245,A -85,B 0,C 180,E1 6779.056,E2 6779.056} C_VEL
LIN {X 0,Y 489.496,Z 706.886,A -85,B 0,C 180,E1 6781.723,E2 6781.723} C_VEL
LIN {X 0,Y 492.64,Z 668.818,A -85,B 0,C 180,E1 6783.93,E2 6783.93} C_VEL
LIN {X 0,Y 495.253,Z 629.206,A -85,B 0,C 180,E1 6785.443,E2 6785.443} C_VEL
LIN {X 0,Y 495.885,Z 593.733,A -85,B 0,C 180,E1 6786.284,E2 6786.284} C_VEL
LIN {X 0,Y 474.751,Z 549.53,A -85,B 0,C 180,E1 6788.886,E2 6788.886} C_VEL
LIN {X 0,Y 474.638,Z 549.53,A -85,B 0,C 180,E1 6795.436,E2 6795.436} C_VEL
LIN {X 0,Y 474.678,Z 549.53,A -85,B 0,C 180,E1 6802.703,E2 6802.703} C_VEL
LIN {X 0,Y 474.828,Z 549.53,A -85,B 0,C 180,E1 6809.42,E2 6809.42} C_VEL
LIN {X 0,Y 474.902,Z 549.53,A -85,B 0,C 180,E1 6815.52,E2 6815.52} C_VEL
LIN {X 0,Y 475.017,Z 549.53,A -85,B 0,C 180,E1 6821.418,E2 6821.418} C_VEL
LIN {X 0,Y 475.176,Z 549.53,A -85,B 0,C 180,E1 6827.116,E2 6827.116} C_VEL
LIN {X 0,Y 475.315,Z 549.53,A -85,B 0,C 180,E1 6832.684,E2 6832.684} C_VEL
LIN {X 0,Y 475.48,Z 549.53,A -85,B 0,C 180,E1 6838.179,E2 6838.179} C_VEL
LIN {X 0,Y 475.433,Z 549.53,A -85,B 0,C 180,E1 6843.655,E2 6843.655} C_VEL
LIN {X 0,Y 475.261,Z 549.53,A -85,B 0,C 180,E1 6849.169,E2 6849.169} C_VEL
LIN {X 0,Y 475.124,Z 549.53,A -85,B 0,C 180,E1 6854.773,E2 6854.773} C_VEL
LIN {X 0,Y 475.01,Z 549.53,A -85,B 0,C 180,E1 6860.529,E2 6860.529} C_VEL
LIN {X 0,Y 474.829,Z 549.53,A -85,B 0,C 180,E1 6866.772,E2 6866.772} C_VEL
LIN {X 0,Y 474.668,Z 549.53,A -85,B 0,C 180,E1 6872.841,E2 6872.841} C_VEL
LIN {X 0,Y 474.713,Z 549.53,A -85,B 0,C 180,E1 6877.304,E2 6877.304} C_VEL
LIN {X 0,Y 474.631,Z 549.53,A -85,B 0,C 180,E1 6882.804,E2 6882.804} C_VEL
LIN {X 0,Y 474.546,Z 549.53,A -85,B 0,C 180,E1 6887.933,E2 6887.933} C_VEL
LIN {X 0,Y 474.724,Z 549.53,A -85,B 0,C 180,E1 6894.965,E2 6894.965} C_VEL
LIN {X 0,Y 474.779,Z 549.53,A -85,B 0,C 180,E1 6901.423,E2 6901.423} C_VEL
LIN {X 0,Y 474.939,Z 549.53,A -85,B 0,C 180,E1 6907.599,E2 6907.599} C_VEL
LIN {X 0,Y 475.103,Z 549.53,A -85,B 0,C 180,E1 6913.334,E2 6913.334} C_VEL
LIN {X 0,Y 475.252,Z 549.53,A -85,B 0,C 180,E1 6918.981,E2 6918.981} C_VEL
LIN {X 0,Y 475.428,Z 549.53,A -85,B 0,C 180,E1 6924.518,E2 6924.518} C_VEL
LIN {X 0,Y 475.605,Z 549.53,A -85,B 0,C 180,E1 6930.001,E2 6930.001} C_VEL
LIN {X 0,Y 475.462,Z 549.53,A -85,B 0,C 180,E1 6935.483,E2 6935.483} C_VEL
LIN {X 0,Y 475.236,Z 549.53,A -85,B 0,C 180,E1 6941.021,E2 6941.021} C_VEL
LIN {X 0,Y 475.075,Z 549.53,A -85,B 0,C 180,E1 6947.032,E2 6947.032} C_VEL
LIN {X 0,Y 475.037,Z 549.53,A -85,B 0,C 180,E1 6952.488,E2 6952.488} C_VEL
LIN {X 0,Y 474.818,Z 549.53,A -85,B 0,C 180,E1 6958.576,E2 6958.576} C_VEL
LIN {X 0,Y 474.712,Z 549.53,A -85,B 0,C 180,E1 6965.037,E2 6965.037} C_VEL
LIN {X 0,Y 474.726,Z 549.53,A -85,B 0,C 180,E1 6967.734,E2 6967.734} C_VEL
LIN {X 0,Y 490.348,Z 589.684,A -85,B 0,C 180,E1 6970.779,E2 6970.779} C_VEL
LIN {X 0,Y 492.409,Z 597.872,A -85,B 0,C 180,E1 6971.392,E2 6971.392} C_VEL
LIN {X 0,Y 489.096,Z 633.437,A -85,B 0,C 180,E1 6973.633,E2 6973.633} C_VEL
LIN {X 0,Y 485.399,Z 666.803,A -85,B 0,C 180,E1 6976.535,E2 6976.535} C_VEL
LIN {X 0,Y 481.891,Z 697.64,A -85,B 0,C 180,E1 6980.116,E2 6980.116} C_VEL
LIN {X 0,Y 479.038,Z 724.781,A -85,B 0,C 180,E1 6984.333,E2 6984.333} C_VEL
LIN {X 0,Y 477.177,Z 746.683,A -85,B 0,C 180,E1 6988.95,E2 6988.95} C_VEL
LIN {X 0,Y 476.175,Z 762.163,A -85,B 0,C 180,E1 6993.564,E2 6993.564} C_VEL
LIN {X 0,Y 475.801,Z 771.047,A -85,B 0,C 180,E1 6997.548,E2 6997.548} C_VEL
LIN {X 0,Y 475.525,Z 776.033,A -85,B 0,C 180,E1 7001.43,E2 7001.43} C_VEL
LIN {X 0,Y 475.507,Z 777.467,A -85,B 0,C 180,E1 7005.239,E2 7005.239} C_VEL
LIN {X 0,Y 475.635,Z 775.57,A -85,B 0,C 180,E1 7008.986,E2 7008.986} C_VEL
LIN {X 0,Y 475.941,Z 768.717,A -85,B 0,C 180,E1 7013.604,E2 7013.604} C_VEL
LIN {X 0,Y 476.481,Z 756.728,A -85,B 0,C 180,E1 7018.175,E2 7018.175} C_VEL
LIN {X 0,Y 477.707,Z 739.158,A -85,B 0,C 180,E1 7022.721,E2 7022.721} C_VEL
LIN {X 0,Y 479.844,Z 716.411,A -85,B 0,C 180,E1 7027.019,E2 7027.019} C_VEL
LIN {X 0,Y 483.015,Z 687.659,A -85,B 0,C 180,E1 7031.065,E2 7031.065} C_VEL
LIN {X 0,Y 486.61,Z 656.072,A -85,B 0,C 180,E1 7034.409,E2 7034.409} C_VEL
LIN {X 0,Y 490.204,Z 622.204,A -85,B 0,C 180,E1 7037.058,E2 7037.058} C_VEL
LIN {X 0,Y 491.866,Z 593.602,A -85,B 0,C 180,E1 7038.757,E2 7038.757} C_VEL
LIN {X 0,Y 477.65,Z 557.055,A -85,B 0,C 180,E1 7041.439,E2 7041.439} C_VEL
LIN {X 0,Y 475.066,Z 549.53,A -85,B 0,C 180,E1 7042.006,E2 7042.006} C_VEL
LIN {X 0,Y 474.789,Z 549.53,A -85,B 0,C 180,E1 7048.572,E2 7048.572} C_VEL
LIN {X 0,Y 474.695,Z 549.53,A -85,B 0,C 180,E1 7055.032,E2 7055.032} C_VEL
LIN {X 0,Y 474.665,Z 549.53,A -85,B 0,C 180,E1 7060.044,E2 7060.044} C_VEL
LIN {X 0,Y 474.633,Z 549.53,A -85,B 0,C 180,E1 7063.171,E2 7063.171} C_VEL
LIN {X 0,Y 470.68,Z 549.53,A -85,B 0,C 180,E1 7065.238,E2 7065.238} C_VEL
LIN {X 0,Y 466.682,Z 549.53,A -85,B 0,C 180,E1 7067.339,E2 7067.339} C_VEL
LIN {X 0,Y 466.782,Z 549.53,A -85,B 0,C 180,E1 7071.008,E2 7071.008} C_VEL
LIN {X 0,Y 487.236,Z 593.844,A -85,B 0,C 180,E1 7073.345,E2 7073.345} C_VEL
LIN {X 0,Y 488.799,Z 597.029,A -85,B 0,C 180,E1 7073.513,E2 7073.513} C_VEL
LIN {X 0,Y 487.159,Z 637.642,A -85,B 0,C 180,E1 7074.528,E2 7074.528} C_VEL
LIN {X 0,Y 484.547,Z 676.799,A -85,B 0,C 180,E1 7076.179,E2 7076.179} C_VEL
LIN {X 0,Y 481.371,Z 713.536,A -85,B 0,C 180,E1 7078.432,E2 7078.432} C_VEL
LIN {X 0,Y 477.89,Z 747.652,A -85,B 0,C 180,E1 7081.286,E2 7081.286} C_VEL
LIN {X 0,Y 474.989,Z 773.963,A -85,B 0,C 180,E1 7084.258,E2 7084.258} C_VEL
LIN {X 0,Y 471.796,Z 801.223,A -85,B 0,C 180,E1 7088.392,E2 7088.392} C_VEL
LIN {X 0,Y 469.694,Z 822.794,A -85,B 0,C 180,E1 7092.773,E2 7092.773} C_VEL
LIN {X 0,Y 468.43,Z 839.279,A -85,B 0,C 180,E1 7097.397,E2 7097.397} C_VEL
LIN {X 0,Y 468.045,Z 849.535,A -85,B 0,C 180,E1 7101.629,E2 7101.629} C_VEL
LIN {X 0,Y 467.8,Z 855.896,A -85,B 0,C 180,E1 7106.288,E2 7106.288} C_VEL
LIN {X 0,Y 467.865,Z 857.5,A -85,B 0,C 180,E1 7109.999,E2 7109.999} C_VEL
LIN {X 0,Y 467.812,Z 855.9,A -85,B 0,C 180,E1 7113.711,E2 7113.711} C_VEL
LIN {X 0,Y 468.073,Z 849.541,A -85,B 0,C 180,E1 7118.369,E2 7118.369} C_VEL
LIN {X 0,Y 468.628,Z 837.901,A -85,B 0,C 180,E1 7123.07,E2 7123.07} C_VEL
LIN {X 0,Y 469.982,Z 819.792,A -85,B 0,C 180,E1 7127.919,E2 7127.919} C_VEL
LIN {X 0,Y 472.208,Z 797.461,A -85,B 0,C 180,E1 7132.249,E2 7132.249} C_VEL
LIN {X 0,Y 475.426,Z 770.15,A -85,B 0,C 180,E1 7136.222,E2 7136.222} C_VEL
LIN {X 0,Y 478.721,Z 741.294,A -85,B 0,C 180,E1 7139.35,E2 7139.35} C_VEL
LIN {X 0,Y 482.354,Z 707.037,A -85,B 0,C 180,E1 7142.138,E2 7142.138} C_VEL
LIN {X 0,Y 485.714,Z 669.37,A -85,B 0,C 180,E1 7144.365,E2 7144.365} C_VEL
LIN {X 0,Y 488.509,Z 630.116,A -85,B 0,C 180,E1 7145.905,E2 7145.905} C_VEL
LIN {X 0,Y 489.349,Z 596.548,A -85,B 0,C 180,E1 7146.733,E2 7146.733} C_VEL
LIN {X 0,Y 466.786,Z 549.53,A -85,B 0,C 180,E1 7149.648,E2 7149.648} C_VEL
LIN {X 0,Y 466.724,Z 549.53,A -85,B 0,C 180,E1 7155.534,E2 7155.534} C_VEL
LIN {X 0,Y 466.66,Z 549.53,A -85,B 0,C 180,E1 7161.949,E2 7161.949} C_VEL
LIN {X 0,Y 466.843,Z 549.53,A -85,B 0,C 180,E1 7168.746,E2 7168.746} C_VEL
LIN {X 0,Y 466.953,Z 549.53,A -85,B 0,C 180,E1 7175.212,E2 7175.212} C_VEL
LIN {X 0,Y 467.065,Z 549.53,A -85,B 0,C 180,E1 7181.09,E2 7181.09} C_VEL
LIN {X 0,Y 467.245,Z 549.53,A -85,B 0,C 180,E1 7186.894,E2 7186.894} C_VEL
LIN {X 0,Y 467.401,Z 549.53,A -85,B 0,C 180,E1 7192.559,E2 7192.559} C_VEL
LIN {X 0,Y 467.576,Z 549.53,A -85,B 0,C 180,E1 7198.148,E2 7198.148} C_VEL
LIN {X 0,Y 467.526,Z 549.53,A -85,B 0,C 180,E1 7203.717,E2 7203.717} C_VEL
LIN {X 0,Y 467.337,Z 549.53,A -85,B 0,C 180,E1 7209.326,E2 7209.326} C_VEL
LIN {X 0,Y 467.193,Z 549.53,A -85,B 0,C 180,E1 7215.03,E2 7215.03} C_VEL
LIN {X 0,Y 467.083,Z 549.53,A -85,B 0,C 180,E1 7220.893,E2 7220.893} C_VEL
LIN {X 0,Y 466.916,Z 549.53,A -85,B 0,C 180,E1 7227.003,E2 7227.003} C_VEL
LIN {X 0,Y 466.737,Z 549.53,A -85,B 0,C 180,E1 7233.472,E2 7233.472} C_VEL
LIN {X 0,Y 466.701,Z 549.53,A -85,B 0,C 180,E1 7240.458,E2 7240.458} C_VEL
LIN {X 0,Y 466.647,Z 549.53,A -85,B 0,C 180,E1 7247.051,E2 7247.051} C_VEL
LIN {X 0,Y 466.65,Z 549.53,A -85,B 0,C 180,E1 7251.943,E2 7251.943} C_VEL
LIN {X 0,Y 466.828,Z 549.53,A -85,B 0,C 180,E1 7258.74,E2 7258.74} C_VEL
LIN {X 0,Y 466.964,Z 549.53,A -85,B 0,C 180,E1 7265.217,E2 7265.217} C_VEL
LIN {X 0,Y 467.093,Z 549.53,A -85,B 0,C 180,E1 7271.087,E2 7271.087} C_VEL
LIN {X 0,Y 467.267,Z 549.53,A -85,B 0,C 180,E1 7276.891,E2 7276.891} C_VEL
LIN {X 0,Y 467.418,Z 549.53,A -85,B 0,C 180,E1 7282.556,E2 7282.556} C_VEL
LIN {X 0,Y 467.64,Z 549.53,A -85,B 0,C 180,E1 7288.145,E2 7288.145} C_VEL
LIN {X 0,Y 467.521,Z 549.53,A -85,B 0,C 180,E1 7293.714,E2 7293.714} C_VEL
LIN {X 0,Y 467.359,Z 549.53,A -85,B 0,C 180,E1 7299.323,E2 7299.323} C_VEL
LIN {X 0,Y 467.219,Z 549.53,A -85,B 0,C 180,E1 7305.026,E2 7305.026} C_VEL
LIN {X 0,Y 467.113,Z 549.53,A -85,B 0,C 180,E1 7310.889,E2 7310.889} C_VEL
LIN {X 0,Y 466.963,Z 549.53,A -85,B 0,C 180,E1 7316.997,E2 7316.997} C_VEL
LIN {X 0,Y 466.782,Z 549.53,A -85,B 0,C 180,E1 7323.465,E2 7323.465} C_VEL
LIN {X 0,Y 466.839,Z 549.672,A -85,B 0,C 180,E1 7327.06,E2 7327.06} C_VEL
LIN {X 0,Y 482.154,Z 588.368,A -85,B 0,C 180,E1 7330.073,E2 7330.073} C_VEL
LIN {X 0,Y 485.484,Z 600.153,A -85,B 0,C 180,E1 7331.011,E2 7331.011} C_VEL
LIN {X 0,Y 481.984,Z 635.454,A -85,B 0,C 180,E1 7333.294,E2 7333.294} C_VEL
LIN {X 0,Y 478.039,Z 669.036,A -85,B 0,C 180,E1 7336.294,E2 7336.294} C_VEL
LIN {X 0,Y 474.248,Z 699.883,A -85,B 0,C 180,E1 7340.016,E2 7340.016} C_VEL
LIN {X 0,Y 471.234,Z 726.647,A -85,B 0,C 180,E1 7344.324,E2 7344.324} C_VEL
LIN {X 0,Y 469.343,Z 747.629,A -85,B 0,C 180,E1 7348.922,E2 7348.922} C_VEL
LIN {X 0,Y 468.3,Z 762.698,A -85,B 0,C 180,E1 7353.566,E2 7353.566} C_VEL
LIN {X 0,Y 467.869,Z 772.261,A -85,B 0,C 180,E1 7358.148,E2 7358.148} C_VEL
LIN {X 0,Y 467.6,Z 777.072,A -85,B 0,C 180,E1 7363.054,E2 7363.054} C_VEL
LIN {X 0,Y 467.618,Z 777.056,A -85,B 0,C 180,E1 7366.897,E2 7366.897} C_VEL
LIN {X 0,Y 467.964,Z 772.47,A -85,B 0,C 180,E1 7371.625,E2 7371.625} C_VEL
LIN {X 0,Y 468.415,Z 762.835,A -85,B 0,C 180,E1 7376.29,E2 7376.29} C_VEL
LIN {X 0,Y 469.325,Z 747.886,A -85,B 0,C 180,E1 7380.92,E2 7380.92} C_VEL
LIN {X 0,Y 471.173,Z 726.963,A -85,B 0,C 180,E1 7385.528,E2 7385.528} C_VEL
LIN {X 0,Y 474.235,Z 700.01,A -85,B 0,C 180,E1 7389.877,E2 7389.877} C_VEL
LIN {X 0,Y 478.114,Z 669.012,A -85,B 0,C 180,E1 7393.618,E2 7393.618} C_VEL
LIN {X 0,Y 481.875,Z 636.334,A -85,B 0,C 180,E1 7396.538,E2 7396.538} C_VEL
LIN {X 0,Y 485.276,Z 600.24,A -85,B 0,C 180,E1 7398.855,E2 7398.855} C_VEL
LIN {X 0,Y 482.426,Z 589.019,A -85,B 0,C 180,E1 7399.687,E2 7399.687} C_VEL
LIN {X 0,Y 467.125,Z 549.53,A -85,B 0,C 180,E1 7402.564,E2 7402.564} C_VEL
LIN {X 0,Y 466.837,Z 549.53,A -85,B 0,C 180,E1 7409.105,E2 7409.105} C_VEL
LIN {X 0,Y 466.733,Z 549.53,A -85,B 0,C 180,E1 7415.806,E2 7415.806} C_VEL
LIN {X 0,Y 466.759,Z 549.53,A -85,B 0,C 180,E1 7421.748,E2 7421.748} C_VEL
LIN {X 0,Y 466.682,Z 549.53,A -85,B 0,C 180,E1 7427.339,E2 7427.339} C_VEL
LIN {X 0,Y 462.676,Z 549.53,A -85,B 0,C 180,E1 7428.711,E2 7428.711} C_VEL
LIN {X 0,Y 458.8,Z 549.53,A -85,B 0,C 180,E1 7430.106,E2 7430.106} C_VEL
LIN {X 0,Y 458.844,Z 550.215,A -85,B 0,C 180,E1 7430.359,E2 7430.359} C_VEL
LIN {X 0,Y 481.902,Z 600.212,A -85,B 0,C 180,E1 7433.111,E2 7433.111} C_VEL
LIN {X 0,Y 479.821,Z 642.703,A -85,B 0,C 180,E1 7434.266,E2 7434.266} C_VEL
LIN {X 0,Y 476.838,Z 683.137,A -85,B 0,C 180,E1 7436.115,E2 7436.115} C_VEL
LIN {X 0,Y 473.184,Z 721.572,A -85,B 0,C 180,E1 7438.685,E2 7438.685} C_VEL
LIN {X 0,Y 469.556,Z 755.238,A -85,B 0,C 180,E1 7441.755,E2 7441.755} C_VEL
LIN {X 0,Y 466.273,Z 784.481,A -85,B 0,C 180,E1 7445.311,E2 7445.311} C_VEL
LIN {X 0,Y 463.245,Z 809.991,A -85,B 0,C 180,E1 7449.679,E2 7449.679} C_VEL
LIN {X 0,Y 461.35,Z 829.826,A -85,B 0,C 180,E1 7454.29,E2 7454.29} C_VEL
LIN {X 0,Y 460.39,Z 844.36,A -85,B 0,C 180,E1 7459.099,E2 7459.099} C_VEL
LIN {X 0,Y 460.04,Z 852.719,A -85,B 0,C 180,E1 7463.385,E2 7463.385} C_VEL
LIN {X 0,Y 459.95,Z 857.085,A -85,B 0,C 180,E1 7468.113,E2 7468.113} C_VEL
LIN {X 0,Y 459.999,Z 857.087,A -85,B 0,C 180,E1 7471.885,E2 7471.885} C_VEL
LIN {X 0,Y 460.046,Z 852.725,A -85,B 0,C 180,E1 7476.614,E2 7476.614} C_VEL
LIN {X 0,Y 460.428,Z 843.216,A -85,B 0,C 180,E1 7481.378,E2 7481.378} C_VEL
LIN {X 0,Y 461.513,Z 828.096,A -85,B 0,C 180,E1 7486.191,E2 7486.191} C_VEL
LIN {X 0,Y 463.663,Z 806.265,A -85,B 0,C 180,E1 7491.05,E2 7491.05} C_VEL
LIN {X 0,Y 466.774,Z 780.835,A -85,B 0,C 180,E1 7495.196,E2 7495.196} C_VEL
LIN {X 0,Y 470.298,Z 749.936,A -85,B 0,C 180,E1 7498.874,E2 7498.874} C_VEL
LIN {X 0,Y 474.168,Z 716.054,A -85,B 0,C 180,E1 7501.909,E2 7501.909} C_VEL
LIN {X 0,Y 477.945,Z 679.163,A -85,B 0,C 180,E1 7504.328,E2 7504.328} C_VEL
LIN {X 0,Y 481.26,Z 639.414,A -85,B 0,C 180,E1 7506.099,E2 7506.099} C_VEL
LIN {X 0,Y 482.669,Z 599.049,A -85,B 0,C 180,E1 7507.211,E2 7507.211} C_VEL
LIN {X 0,Y 458.858,Z 549.53,A -85,B 0,C 180,E1 7510.303,E2 7510.303} C_VEL
LIN {X 0,Y 458.792,Z 549.53,A -85,B 0,C 180,E1 7516.553,E2 7516.553} C_VEL
LIN {X 0,Y 458.76,Z 549.53,A -85,B 0,C 180,E1 7523.56,E2 7523.56} C_VEL
LIN {X 0,Y 458.899,Z 549.53,A -85,B 0,C 180,E1 7530.342,E2 7530.342} C_VEL
LIN {X 0,Y 459.03,Z 549.53,A -85,B 0,C 180,E1 7536.689,E2 7536.689} C_VEL
LIN {X 0,Y 459.251,Z 549.53,A -85,B 0,C 180,E1 7542.953,E2 7542.953} C_VEL
LIN {X 0,Y 459.37,Z 549.53,A -85,B 0,C 180,E1 7548.598,E2 7548.598} C_VEL
LIN {X 0,Y 459.561,Z 549.53,A -85,B 0,C 180,E1 7554.332,E2 7554.332} C_VEL
LIN {X 0,Y 459.756,Z 549.53,A -85,B 0,C 180,E1 7560.004,E2 7560.004} C_VEL
LIN {X 0,Y 459.613,Z 549.53,A -85,B 0,C 180,E1 7565.675,E2 7565.675} C_VEL
LIN {X 0,Y 459.356,Z 549.53,A -85,B 0,C 180,E1 7571.41,E2 7571.41} C_VEL
LIN {X 0,Y 459.239,Z 549.53,A -85,B 0,C 180,E1 7577.264,E2 7577.264} C_VEL
LIN {X 0,Y 459.091,Z 549.53,A -85,B 0,C 180,E1 7583.317,E2 7583.317} C_VEL
LIN {X 0,Y 458.853,Z 549.53,A -85,B 0,C 180,E1 7589.67,E2 7589.67} C_VEL
LIN {X 0,Y 458.757,Z 549.53,A -85,B 0,C 180,E1 7596.45,E2 7596.45} C_VEL
LIN {X 0,Y 458.807,Z 549.53,A -85,B 0,C 180,E1 7601.304,E2 7601.304} C_VEL
LIN {X 0,Y 458.726,Z 549.53,A -85,B 0,C 180,E1 7606.567,E2 7606.567} C_VEL
LIN {X 0,Y 458.753,Z 549.53,A -85,B 0,C 180,E1 7613.555,E2 7613.555} C_VEL
LIN {X 0,Y 458.881,Z 549.53,A -85,B 0,C 180,E1 7620.336,E2 7620.336} C_VEL
LIN {X 0,Y 459.048,Z 549.53,A -85,B 0,C 180,E1 7626.685,E2 7626.685} C_VEL
LIN {X 0,Y 459.268,Z 549.53,A -85,B 0,C 180,E1 7632.957,E2 7632.957} C_VEL
LIN {X 0,Y 459.394,Z 549.53,A -85,B 0,C 180,E1 7638.596,E2 7638.596} C_VEL
LIN {X 0,Y 459.593,Z 549.53,A -85,B 0,C 180,E1 7644.329,E2 7644.329} C_VEL
LIN {X 0,Y 459.817,Z 549.53,A -85,B 0,C 180,E1 7650.001,E2 7650.001} C_VEL
LIN {X 0,Y 459.63,Z 549.53,A -85,B 0,C 180,E1 7655.672,E2 7655.672} C_VEL
LIN {X 0,Y 459.38,Z 549.53,A -85,B 0,C 180,E1 7661.406,E2 7661.406} C_VEL
LIN {X 0,Y 459.253,Z 549.53,A -85,B 0,C 180,E1 7667.261,E2 7667.261} C_VEL
LIN {X 0,Y 459.141,Z 549.53,A -85,B 0,C 180,E1 7673.311,E2 7673.311} C_VEL
LIN {X 0,Y 458.884,Z 549.53,A -85,B 0,C 180,E1 7679.665,E2 7679.665} C_VEL
LIN {X 0,Y 458.858,Z 549.53,A -85,B 0,C 180,E1 7686.304,E2 7686.304} C_VEL
LIN {X 0,Y 474.57,Z 588.802,A -85,B 0,C 180,E1 7689.486,E2 7689.486} C_VEL
LIN {X 0,Y 478.594,Z 602.083,A -85,B 0,C 180,E1 7690.597,E2 7690.597} C_VEL
LIN {X 0,Y 474.807,Z 638.04,A -85,B 0,C 180,E1 7692.991,E2 7692.991} C_VEL
LIN {X 0,Y 470.654,Z 671.456,A -85,B 0,C 180,E1 7696.064,E2 7696.064} C_VEL
LIN {X 0,Y 466.712,Z 701.43,A -85,B 0,C 180,E1 7699.802,E2 7699.802} C_VEL
LIN {X 0,Y 463.496,Z 727.954,A -85,B 0,C 180,E1 7704.227,E2 7704.227} C_VEL
LIN {X 0,Y 461.443,Z 749.039,A -85,B 0,C 180,E1 7709.015,E2 7709.015} C_VEL
LIN {X 0,Y 460.396,Z 763.39,A -85,B 0,C 180,E1 7713.639,E2 7713.639} C_VEL
LIN {X 0,Y 459.977,Z 772.137,A -85,B 0,C 180,E1 7717.954,E2 7717.954} C_VEL
LIN {X 0,Y 459.674,Z 776.982,A -85,B 0,C 180,E1 7722.787,E2 7722.787} C_VEL
LIN {X 0,Y 459.709,Z 777.154,A -85,B 0,C 180,E1 7726.667,E2 7726.667} C_VEL
LIN {X 0,Y 460.078,Z 772.585,A -85,B 0,C 180,E1 7731.656,E2 7731.656} C_VEL
LIN {X 0,Y 460.557,Z 762.267,A -85,B 0,C 180,E1 7736.698,E2 7736.698} C_VEL
LIN {X 0,Y 461.588,Z 747.096,A -85,B 0,C 180,E1 7741.406,E2 7741.406} C_VEL
LIN {X 0,Y 463.677,Z 725.853,A -85,B 0,C 180,E1 7746.088,E2 7746.088} C_VEL
LIN {X 0,Y 467.084,Z 698.776,A -85,B 0,C 180,E1 7750.502,E2 7750.502} C_VEL
LIN {X 0,Y 470.972,Z 669.448,A -85,B 0,C 180,E1 7754.066,E2 7754.066} C_VEL
LIN {X 0,Y 474.869,Z 637.365,A -85,B 0,C 180,E1 7756.956,E2 7756.956} C_VEL
LIN {X 0,Y 478.436,Z 601.012,A -85,B 0,C 180,E1 7759.312,E2 7759.312} C_VEL
LIN {X 0,Y 464.842,Z 563.765,A -85,B 0,C 180,E1 7762.233,E2 7762.233} C_VEL
LIN {X 0,Y 459.111,Z 549.53,A -85,B 0,C 180,E1 7763.307,E2 7763.307} C_VEL
LIN {X 0,Y 458.857,Z 549.53,A -85,B 0,C 180,E1 7769.661,E2 7769.661} C_VEL
LIN {X 0,Y 458.774,Z 549.53,A -85,B 0,C 180,E1 7776.438,E2 7776.438} C_VEL
LIN {X 0,Y 458.851,Z 549.53,A -85,B 0,C 180,E1 7781.288,E2 7781.288} C_VEL
LIN {X 0,Y 458.696,Z 549.53,A -85,B 0,C 180,E1 7787.329,E2 7787.329} C_VEL
LIN {X 0,Y 458.8,Z 549.53,A -85,B 0,C 180,E1 7790.106,E2 7790.106} C_VEL
LIN {X 0,Y 460.897,Z 552.351,A -85,B 0,C 180,E1 7790.582,E2 7790.582} C_VEL
LIN {X 0,Y 463.525,Z 563.291,A -85,B 0,C 180,E1 7791.005,E2 7791.005} C_VEL
LIN {X 0,Y 464.876,Z 581.004,A -85,B 0,C 180,E1 7791.476,E2 7791.476} C_VEL
LIN {X 0,Y 465.27,Z 582.15,A -85,B 0,C 180,E1 7791.531,E2 7791.531} C_VEL
LIN {X 0,Y 475,Z 602.034,A -85,B 0,C 180,E1 7792.666,E2 7792.666} C_VEL
LIN {X 0,Y 472.633,Z 645.318,A -85,B 0,C 180,E1 7793.921,E2 7793.921} C_VEL
LIN {X 0,Y 469.402,Z 685.45,A -85,B 0,C 180,E1 7795.849,E2 7795.849} C_VEL
LIN {X 0,Y 465.782,Z 721.569,A -85,B 0,C 180,E1 7798.333,E2 7798.333} C_VEL
LIN {X 0,Y 461.958,Z 755.332,A -85,B 0,C 180,E1 7801.475,E2 7801.475} C_VEL
LIN {X 0,Y 458.509,Z 785.038,A -85,B 0,C 180,E1 7805.151,E2 7805.151} C_VEL
LIN {X 0,Y 455.9,Z 807.574,A -85,B 0,C 180,E1 7808.827,E2 7808.827} C_VEL
LIN {X 0,Y 453.719,Z 828.088,A -85,B 0,C 180,E1 7813.521,E2 7813.521} C_VEL
LIN {X 0,Y 452.553,Z 843.213,A -85,B 0,C 180,E1 7818.419,E2 7818.419} C_VEL
LIN {X 0,Y 452.148,Z 852.718,A -85,B 0,C 180,E1 7823.269,E2 7823.269} C_VEL
LIN {X 0,Y 452.047,Z 857.085,A -85,B 0,C 180,E1 7828.08,E2 7828.08} C_VEL
LIN {X 0,Y 452.124,Z 857.087,A -85,B 0,C 180,E1 7831.918,E2 7831.918} C_VEL
LIN {X 0,Y 452.152,Z 852.725,A -85,B 0,C 180,E1 7836.73,E2 7836.73} C_VEL
LIN {X 0,Y 452.569,Z 843.216,A -85,B 0,C 180,E1 7841.579,E2 7841.579} C_VEL
LIN {X 0,Y 453.779,Z 828.096,A -85,B 0,C 180,E1 7846.475,E2 7846.475} C_VEL
LIN {X 0,Y 456.107,Z 806.261,A -85,B 0,C 180,E1 7851.416,E2 7851.416} C_VEL
LIN {X 0,Y 459.267,Z 779.832,A -85,B 0,C 180,E1 7855.638,E2 7855.638} C_VEL
LIN {X 0,Y 463.083,Z 748.823,A -85,B 0,C 180,E1 7859.368,E2 7859.368} C_VEL
LIN {X 0,Y 467.104,Z 715.505,A -85,B 0,C 180,E1 7862.388,E2 7862.388} C_VEL
LIN {X 0,Y 471.061,Z 679.08,A -85,B 0,C 180,E1 7864.812,E2 7864.812} C_VEL
LIN {X 0,Y 474.527,Z 639.905,A -85,B 0,C 180,E1 7866.593,E2 7866.593} C_VEL
LIN {X 0,Y 476.032,Z 601.689,A -85,B 0,C 180,E1 7867.695,E2 7867.695} C_VEL
LIN {X 0,Y 450.984,Z 549.53,A -85,B 0,C 180,E1 7871.084,E2 7871.084} C_VEL
LIN {X 0,Y 450.766,Z 549.53,A -85,B 0,C 180,E1 7877.803,E2 7877.803} C_VEL
LIN {X 0,Y 450.859,Z 549.53,A -85,B 0,C 180,E1 7883.702,E2 7883.702} C_VEL
LIN {X 0,Y 450.988,Z 549.53,A -85,B 0,C 180,E1 7889.768,E2 7889.768} C_VEL
LIN {X 0,Y 451.07,Z 549.53,A -85,B 0,C 180,E1 7896.252,E2 7896.252} C_VEL
LIN {X 0,Y 451.265,Z 549.53,A -85,B 0,C 180,E1 7902.429,E2 7902.429} C_VEL
LIN {X 0,Y 451.44,Z 549.53,A -85,B 0,C 180,E1 7908.395,E2 7908.395} C_VEL
LIN {X 0,Y 451.646,Z 549.53,A -85,B 0,C 180,E1 7914.232,E2 7914.232} C_VEL
LIN {X 0,Y 451.856,Z 549.53,A -85,B 0,C 180,E1 7920.004,E2 7920.004} C_VEL
LIN {X 0,Y 451.726,Z 549.53,A -85,B 0,C 180,E1 7925.775,E2 7925.775} C_VEL
LIN {X 0,Y 451.428,Z 549.53,A -85,B 0,C 180,E1 7931.613,E2 7931.613} C_VEL
LIN {X 0,Y 451.296,Z 549.53,A -85,B 0,C 180,E1 7937.578,E2 7937.578} C_VEL
LIN {X 0,Y 451.124,Z 549.53,A -85,B 0,C 180,E1 7943.754,E2 7943.754} C_VEL
LIN {X 0,Y 450.922,Z 549.53,A -85,B 0,C 180,E1 7950.246,E2 7950.246} C_VEL
LIN {X 0,Y 450.867,Z 549.53,A -85,B 0,C 180,E1 7957.194,E2 7957.194} C_VEL
LIN {X 0,Y 450.831,Z 549.53,A -85,B 0,C 180,E1 7962.368,E2 7962.368} C_VEL
LIN {X 0,Y 450.73,Z 549.53,A -85,B 0,C 180,E1 7967.793,E2 7967.793} C_VEL
LIN {X 0,Y 450.855,Z 549.53,A -85,B 0,C 180,E1 7973.709,E2 7973.709} C_VEL
LIN {X 0,Y 450.963,Z 549.53,A -85,B 0,C 180,E1 7979.762,E2 7979.762} C_VEL
LIN {X 0,Y 451.083,Z 549.53,A -85,B 0,C 180,E1 7986.249,E2 7986.249} C_VEL
LIN {X 0,Y 451.303,Z 549.53,A -85,B 0,C 180,E1 7992.427,E2 7992.427} C_VEL
LIN {X 0,Y 451.465,Z 549.53,A -85,B 0,C 180,E1 7998.393,E2 7998.393} C_VEL
LIN {X 0,Y 451.676,Z 549.53,A -85,B 0,C 180,E1 8004.229,E2 8004.229} C_VEL
LIN {X 0,Y 451.947,Z 549.53,A -85,B 0,C 180,E1 8010.001,E2 8010.001} C_VEL
LIN {X 0,Y 451.744,Z 549.53,A -85,B 0,C 180,E1 8015.772,E2 8015.772} C_VEL
LIN {X 0,Y 451.451,Z 549.53,A -85,B 0,C 180,E1 8021.61,E2 8021.61} C_VEL
LIN {X 0,Y 451.312,Z 549.53,A -85,B 0,C 180,E1 8027.575,E2 8027.575} C_VEL
LIN {X 0,Y 451.179,Z 549.53,A -85,B 0,C 180,E1 8033.748,E2 8033.748} C_VEL
LIN {X 0,Y 450.954,Z 549.53,A -85,B 0,C 180,E1 8040.241,E2 8040.241} C_VEL
LIN {X 0,Y 450.993,Z 550.268,A -85,B 0,C 180,E1 8045.608,E2 8045.608} C_VEL
LIN {X 0,Y 466.024,Z 586.791,A -85,B 0,C 180,E1 8048.651,E2 8048.651} C_VEL
LIN {X 0,Y 471.614,Z 605.362,A -85,B 0,C 180,E1 8050.25,E2 8050.25} C_VEL
LIN {X 0,Y 467.569,Z 641.122,A -85,B 0,C 180,E1 8052.717,E2 8052.717} C_VEL
LIN {X 0,Y 463.286,Z 673.937,A -85,B 0,C 180,E1 8055.837,E2 8055.837} C_VEL
LIN {X 0,Y 459.035,Z 704.523,A -85,B 0,C 180,E1 8059.786,E2 8059.786} C_VEL
LIN {X 0,Y 455.647,Z 729.934,A -85,B 0,C 180,E1 8064.261,E2 8064.261} C_VEL
LIN {X 0,Y 453.587,Z 749.913,A -85,B 0,C 180,E1 8068.976,E2 8068.976} C_VEL
LIN {X 0,Y 452.518,Z 763.99,A -85,B 0,C 180,E1 8073.693,E2 8073.693} C_VEL
LIN {X 0,Y 452.033,Z 772.915,A -85,B 0,C 180,E1 8078.377,E2 8078.377} C_VEL
LIN {X 0,Y 451.766,Z 776.824,A -85,B 0,C 180,E1 8082.441,E2 8082.441} C_VEL
LIN {X 0,Y 451.803,Z 777.252,A -85,B 0,C 180,E1 8086.429,E2 8086.429} C_VEL
LIN {X 0,Y 452.187,Z 772.789,A -85,B 0,C 180,E1 8091.622,E2 8091.622} C_VEL
LIN {X 0,Y 452.688,Z 762.959,A -85,B 0,C 180,E1 8096.641,E2 8096.641} C_VEL
LIN {X 0,Y 453.756,Z 748.08,A -85,B 0,C 180,E1 8101.43,E2 8101.43} C_VEL
LIN {X 0,Y 455.932,Z 727.318,A -85,B 0,C 180,E1 8106.192,E2 8106.192} C_VEL
LIN {X 0,Y 459.353,Z 702.592,A -85,B 0,C 180,E1 8110.44,E2 8110.44} C_VEL
LIN {X 0,Y 463.263,Z 674.199,A -85,B 0,C 180,E1 8114.064,E2 8114.064} C_VEL
LIN {X 0,Y 467.433,Z 642.125,A -85,B 0,C 180,E1 8117.089,E2 8117.089} C_VEL
LIN {X 0,Y 471.071,Z 607.318,A -85,B 0,C 180,E1 8119.475,E2 8119.475} C_VEL
LIN {X 0,Y 470.569,Z 599.865,A -85,B 0,C 180,E1 8119.987,E2 8119.987} C_VEL
LIN {X 0,Y 455.466,Z 560.095,A -85,B 0,C 180,E1 8123.195,E2 8123.195} C_VEL
LIN {X 0,Y 451.147,Z 549.53,A -85,B 0,C 180,E1 8124.061,E2 8124.061} C_VEL
LIN {X 0,Y 450.928,Z 549.53,A -85,B 0,C 180,E1 8130.236,E2 8130.236} C_VEL
LIN {X 0,Y 450.878,Z 549.53,A -85,B 0,C 180,E1 8137.183,E2 8137.183} C_VEL
LIN {X 0,Y 450.866,Z 549.53,A -85,B 0,C 180,E1 8142.371,E2 8142.371} C_VEL
LIN {X 0,Y 450.83,Z 549.53,A -85,B 0,C 180,E1 8149.305,E2 8149.305} C_VEL
LIN {X 0,Y 450.907,Z 550.244,A -85,B 0,C 180,E1 8149.629,E2 8149.629} C_VEL
LIN {X 0,Y 465.27,Z 582.15,A -85,B 0,C 180,E1 8151.531,E2 8151.531} C_VEL
LIN {X 0,Y 467.473,Z 593.292,A -85,B 0,C 180,E1 8151.918,E2 8151.918} C_VEL
LIN {X 0,Y 468.023,Z 604.985,A -85,B 0,C 180,E1 8152.232,E2 8152.232} C_VEL
LIN {X 0,Y 465.49,Z 647.172,A -85,B 0,C 180,E1 8153.544,E2 8153.544} C_VEL
LIN {X 0,Y 462.099,Z 686.603,A -85,B 0,C 180,E1 8155.507,E2 8155.507} C_VEL
LIN {X 0,Y 458.242,Z 722.961,A -85,B 0,C 180,E1 8158.085,E2 8158.085} C_VEL
LIN {X 0,Y 454.218,Z 757.081,A -85,B 0,C 180,E1 8161.368,E2 8161.368} C_VEL
LIN {X 0,Y 450.651,Z 786.203,A -85,B 0,C 180,E1 8165.098,E2 8165.098} C_VEL
LIN {X 0,Y 447.797,Z 810.514,A -85,B 0,C 180,E1 8169.204,E2 8169.204} C_VEL
LIN {X 0,Y 445.957,Z 828.088,A -85,B 0,C 180,E1 8173.226,E2 8173.226} C_VEL
LIN {X 0,Y 444.692,Z 843.213,A -85,B 0,C 180,E1 8178.211,E2 8178.211} C_VEL
LIN {X 0,Y 444.266,Z 852.718,A -85,B 0,C 180,E1 8183.149,E2 8183.149} C_VEL
LIN {X 0,Y 444.142,Z 857.086,A -85,B 0,C 180,E1 8188.046,E2 8188.046} C_VEL
LIN {X 0,Y 444.217,Z 857.087,A -85,B 0,C 180,E1 8191.952,E2 8191.952} C_VEL
LIN {X 0,Y 444.27,Z 852.725,A -85,B 0,C 180,E1 8196.85,E2 8196.85} C_VEL
LIN {X 0,Y 444.721,Z 843.216,A -85,B 0,C 180,E1 8201.786,E2 8201.786} C_VEL
LIN {X 0,Y 446.036,Z 828.096,A -85,B 0,C 180,E1 8206.769,E2 8206.769} C_VEL
LIN {X 0,Y 447.967,Z 809.402,A -85,B 0,C 180,E1 8211.045,E2 8211.045} C_VEL
LIN {X 0,Y 451.147,Z 784.296,A -85,B 0,C 180,E1 8215.305,E2 8215.305} C_VEL
LIN {X 0,Y 455.243,Z 752.485,A -85,B 0,C 180,E1 8219.377,E2 8219.377} C_VEL
LIN {X 0,Y 459.667,Z 718.254,A -85,B 0,C 180,E1 8222.622,E2 8222.622} C_VEL
LIN {X 0,Y 464.046,Z 680.558,A -85,B 0,C 180,E1 8225.222,E2 8225.222} C_VEL
LIN {X 0,Y 467.773,Z 641.387,A -85,B 0,C 180,E1 8227.062,E2 8227.062} C_VEL
LIN {X 0,Y 469.611,Z 604.567,A -85,B 0,C 180,E1 8228.17,E2 8228.17} C_VEL
LIN {X 0,Y 444.269,Z 553.793,A -85,B 0,C 180,E1 8231.625,E2 8231.625} C_VEL
LIN {X 0,Y 442.986,Z 549.53,A -85,B 0,C 180,E1 8231.998,E2 8231.998} C_VEL
LIN {X 0,Y 442.788,Z 549.53,A -85,B 0,C 180,E1 8238.786,E2 8238.786} C_VEL
LIN {X 0,Y 442.965,Z 549.53,A -85,B 0,C 180,E1 8245.116,E2 8245.116} C_VEL
LIN {X 0,Y 443.055,Z 549.53,A -85,B 0,C 180,E1 8251.423,E2 8251.423} C_VEL
LIN {X 0,Y 443.175,Z 549.53,A -85,B 0,C 180,E1 8257.931,E2 8257.931} C_VEL
LIN {X 0,Y 443.39,Z 549.53,A -85,B 0,C 180,E1 8264.151,E2 8264.151} C_VEL
LIN {X 0,Y 443.648,Z 549.53,A -85,B 0,C 180,E1 8270.18,E2 8270.18} C_VEL
LIN {X 0,Y 443.852,Z 549.53,A -85,B 0,C 180,E1 8276.092,E2 8276.092} C_VEL
LIN {X 0,Y 444.05,Z 549.53,A -85,B 0,C 180,E1 8281.958,E2 8281.958} C_VEL
LIN {X 0,Y 443.665,Z 549.53,A -85,B 0,C 180,E1 8288.251,E2 8288.251} C_VEL
LIN {X 0,Y 443.471,Z 549.53,A -85,B 0,C 180,E1 8293.831,E2 8293.831} C_VEL
LIN {X 0,Y 443.325,Z 549.53,A -85,B 0,C 180,E1 8299.974,E2 8299.974} C_VEL
LIN {X 0,Y 443.118,Z 549.53,A -85,B 0,C 180,E1 8306.375,E2 8306.375} C_VEL
LIN {X 0,Y 442.911,Z 549.53,A -85,B 0,C 180,E1 8313.162,E2 8313.162} C_VEL
LIN {X 0,Y 442.883,Z 549.53,A -85,B 0,C 180,E1 8318.161,E2 8318.161} C_VEL
LIN {X 0,Y 442.82,Z 549.53,A -85,B 0,C 180,E1 8324.11,E2 8324.11} C_VEL
LIN {X 0,Y 442.771,Z 549.53,A -85,B 0,C 180,E1 8329.481,E2 8329.481} C_VEL
LIN {X 0,Y 442.967,Z 549.53,A -85,B 0,C 180,E1 8335.122,E2 8335.122} C_VEL
LIN {X 0,Y 443.027,Z 549.53,A -85,B 0,C 180,E1 8341.416,E2 8341.416} C_VEL
LIN {X 0,Y 443.199,Z 549.53,A -85,B 0,C 180,E1 8347.928,E2 8347.928} C_VEL
LIN {X 0,Y 443.42,Z 549.53,A -85,B 0,C 180,E1 8354.148,E2 8354.148} C_VEL
LIN {X 0,Y 443.674,Z 549.53,A -85,B 0,C 180,E1 8360.177,E2 8360.177} C_VEL
LIN {X 0,Y 443.981,Z 549.53,A -85,B 0,C 180,E1 8366.09,E2 8366.09} C_VEL
LIN {X 0,Y 444.052,Z 549.53,A -85,B 0,C 180,E1 8371.955,E2 8371.955} C_VEL
LIN {X 0,Y 443.666,Z 549.53,A -85,B 0,C 180,E1 8378.228,E2 8378.228} C_VEL
LIN {X 0,Y 443.491,Z 549.53,A -85,B 0,C 180,E1 8383.827,E2 8383.827} C_VEL
LIN {X 0,Y 443.352,Z 549.53,A -85,B 0,C 180,E1 8389.969,E2 8389.969} C_VEL
LIN {X 0,Y 443.171,Z 549.53,A -85,B 0,C 180,E1 8396.369,E2 8396.369} C_VEL
LIN {X 0,Y 442.927,Z 549.53,A -85,B 0,C 180,E1 8403.572,E2 8403.572} C_VEL
LIN {X 0,Y 443.03,Z 550.084,A -85,B 0,C 180,E1 8404.816,E2 8404.816} C_VEL
LIN {X 0,Y 458.747,Z 587.956,A -85,B 0,C 180,E1 8408.082,E2 8408.082} C_VEL
LIN {X 0,Y 464.814,Z 607.165,A -85,B 0,C 180,E1 8409.809,E2 8409.809} C_VEL
LIN {X 0,Y 460.513,Z 643.036,A -85,B 0,C 180,E1 8412.342,E2 8412.342} C_VEL
LIN {X 0,Y 455.904,Z 676.445,A -85,B 0,C 180,E1 8415.611,E2 8415.611} C_VEL
LIN {X 0,Y 451.587,Z 705.783,A -85,B 0,C 180,E1 8419.501,E2 8419.501} C_VEL
LIN {X 0,Y 448.111,Z 730.398,A -85,B 0,C 180,E1 8423.913,E2 8423.913} C_VEL
LIN {X 0,Y 445.697,Z 751.066,A -85,B 0,C 180,E1 8429.029,E2 8429.029} C_VEL
LIN {X 0,Y 444.622,Z 764.529,A -85,B 0,C 180,E1 8433.721,E2 8433.721} C_VEL
LIN {X 0,Y 444.179,Z 772.533,A -85,B 0,C 180,E1 8437.975,E2 8437.975} C_VEL
LIN {X 0,Y 443.84,Z 777.006,A -85,B 0,C 180,E1 8442.78,E2 8442.78} C_VEL
LIN {X 0,Y 443.88,Z 777.344,A -85,B 0,C 180,E1 8446.182,E2 8446.182} C_VEL
LIN {X 0,Y 444.229,Z 773.311,A -85,B 0,C 180,E1 8451.347,E2 8451.347} C_VEL
LIN {X 0,Y 444.823,Z 763.609,A -85,B 0,C 180,E1 8456.581,E2 8456.581} C_VEL
LIN {X 0,Y 445.905,Z 749.066,A -85,B 0,C 180,E1 8461.455,E2 8461.455} C_VEL
LIN {X 0,Y 448.445,Z 728.021,A -85,B 0,C 180,E1 8466.539,E2 8466.539} C_VEL
LIN {X 0,Y 452.068,Z 703.183,A -85,B 0,C 180,E1 8470.855,E2 8470.855} C_VEL
LIN {X 0,Y 456.221,Z 674.592,A -85,B 0,C 180,E1 8474.531,E2 8474.531} C_VEL
LIN {X 0,Y 460.471,Z 643.099,A -85,B 0,C 180,E1 8477.53,E2 8477.53} C_VEL
LIN {X 0,Y 464.272,Z 608.088,A -85,B 0,C 180,E1 8479.959,E2 8479.959} C_VEL
LIN {X 0,Y 462.705,Z 599.728,A -85,B 0,C 180,E1 8480.62,E2 8480.62} C_VEL
LIN {X 0,Y 448.4,Z 562.043,A -85,B 0,C 180,E1 8483.787,E2 8483.787} C_VEL
LIN {X 0,Y 443.236,Z 549.53,A -85,B 0,C 180,E1 8484.798,E2 8484.798} C_VEL
LIN {X 0,Y 442.933,Z 549.53,A -85,B 0,C 180,E1 8491.286,E2 8491.286} C_VEL
LIN {X 0,Y 442.906,Z 549.53,A -85,B 0,C 180,E1 8497.969,E2 8497.969} C_VEL
LIN {X 0,Y 442.885,Z 549.53,A -85,B 0,C 180,E1 8504.116,E2 8504.116} C_VEL
LIN {X 0,Y 442.958,Z 550.26,A -85,B 0,C 180,E1 8508.838,E2 8508.838} C_VEL
LIN {X 0,Y 468.023,Z 604.985,A -85,B 0,C 180,E1 8512.232,E2 8512.232} C_VEL
LIN {X 0,Y 465.644,Z 617.717,A -85,B 0,C 180,E1 8512.421,E2 8512.421} C_VEL
LIN {X 0,Y 459.45,Z 636.55,A -85,B 0,C 180,E1 8512.668,E2 8512.668} C_VEL
LIN {X 0,Y 459.233,Z 638.674,A -85,B 0,C 180,E1 8512.74,E2 8512.74} C_VEL
LIN {X 0,Y 455.632,Z 680.158,A -85,B 0,C 180,E1 8514.693,E2 8514.693} C_VEL
LIN {X 0,Y 451.439,Z 718.618,A -85,B 0,C 180,E1 8517.35,E2 8517.35} C_VEL
LIN {X 0,Y 447.145,Z 752.904,A -85,B 0,C 180,E1 8520.594,E2 8520.594} C_VEL
LIN {X 0,Y 443.245,Z 783.686,A -85,B 0,C 180,E1 8524.496,E2 8524.496} C_VEL
LIN {X 0,Y 440.148,Z 808.885,A -85,B 0,C 180,E1 8528.748,E2 8528.748} C_VEL
LIN {X 0,Y 438.201,Z 827.517,A -85,B 0,C 180,E1 8532.92,E2 8532.92} C_VEL
LIN {X 0,Y 436.926,Z 841.952,A -85,B 0,C 180,E1 8537.491,E2 8537.491} C_VEL
LIN {X 0,Y 436.431,Z 851.175,A -85,B 0,C 180,E1 8542.023,E2 8542.023} C_VEL
LIN {X 0,Y 436.207,Z 855.894,A -85,B 0,C 180,E1 8546.018,E2 8546.018} C_VEL
LIN {X 0,Y 436.271,Z 857.5,A -85,B 0,C 180,E1 8549.999,E2 8549.999} C_VEL
LIN {X 0,Y 436.227,Z 855.899,A -85,B 0,C 180,E1 8553.98,E2 8553.98} C_VEL
LIN {X 0,Y 436.579,Z 849.25,A -85,B 0,C 180,E1 8559.13,E2 8559.13} C_VEL
LIN {X 0,Y 437.462,Z 837.017,A -85,B 0,C 180,E1 8564.307,E2 8564.307} C_VEL
LIN {X 0,Y 439.038,Z 819.56,A -85,B 0,C 180,E1 8569.067,E2 8569.067} C_VEL
LIN {X 0,Y 441.948,Z 795.987,A -85,B 0,C 180,E1 8573.736,E2 8573.736} C_VEL
LIN {X 0,Y 445.758,Z 768.078,A -85,B 0,C 180,E1 8577.882,E2 8577.882} C_VEL
LIN {X 0,Y 450.061,Z 737.177,A -85,B 0,C 180,E1 8581.365,E2 8581.365} C_VEL
LIN {X 0,Y 454.716,Z 702.474,A -85,B 0,C 180,E1 8584.29,E2 8584.29} C_VEL
LIN {X 0,Y 458.822,Z 666.203,A -85,B 0,C 180,E1 8586.505,E2 8586.505} C_VEL
LIN {X 0,Y 462.243,Z 626.806,A -85,B 0,C 180,E1 8588.107,E2 8588.107} C_VEL
LIN {X 0,Y 462.941,Z 606.937,A -85,B 0,C 180,E1 8588.692,E2 8588.692} C_VEL
LIN {X 0,Y 437.163,Z 554.873,A -85,B 0,C 180,E1 8592.332,E2 8592.332} C_VEL
LIN {X 0,Y 435.014,Z 549.53,A -85,B 0,C 180,E1 8592.791,E2 8592.791} C_VEL
LIN {X 0,Y 434.885,Z 549.53,A -85,B 0,C 180,E1 8598.593,E2 8598.593} C_VEL
LIN {X 0,Y 434.922,Z 549.53,A -85,B 0,C 180,E1 8603.721,E2 8603.721} C_VEL
LIN {X 0,Y 435.089,Z 549.53,A -85,B 0,C 180,E1 8608.54,E2 8608.54} C_VEL
LIN {X 0,Y 435.183,Z 549.53,A -85,B 0,C 180,E1 8615.329,E2 8615.329} C_VEL
LIN {X 0,Y 435.391,Z 549.53,A -85,B 0,C 180,E1 8621.766,E2 8621.766} C_VEL
LIN {X 0,Y 435.585,Z 549.53,A -85,B 0,C 180,E1 8627.967,E2 8627.967} C_VEL
LIN {X 0,Y 435.814,Z 549.53,A -85,B 0,C 180,E1 8634.022,E2 8634.022} C_VEL
LIN {X 0,Y 436.068,Z 549.53,A -85,B 0,C 180,E1 8640.004,E2 8640.004} C_VEL
LIN {X 0,Y 435.887,Z 549.53,A -85,B 0,C 180,E1 8645.985,E2 8645.985} C_VEL
LIN {X 0,Y 435.578,Z 549.53,A -85,B 0,C 180,E1 8652.042,E2 8652.042} C_VEL
LIN {X 0,Y 435.426,Z 549.53,A -85,B 0,C 180,E1 8658.241,E2 8658.241} C_VEL
LIN {X 0,Y 435.224,Z 549.53,A -85,B 0,C 180,E1 8664.678,E2 8664.678} C_VEL
LIN {X 0,Y 435.012,Z 549.53,A -85,B 0,C 180,E1 8671.476,E2 8671.476} C_VEL
LIN {X 0,Y 434.91,Z 549.53,A -85,B 0,C 180,E1 8678.807,E2 8678.807} C_VEL
LIN {X 0,Y 434.917,Z 549.53,A -85,B 0,C 180,E1 8684.132,E2 8684.132} C_VEL
LIN {X 0,Y 434.847,Z 549.53,A -85,B 0,C 180,E1 8691.192,E2 8691.192} C_VEL
LIN {X 0,Y 435.08,Z 549.53,A -85,B 0,C 180,E1 8696.641,E2 8696.641} C_VEL
LIN {X 0,Y 435.138,Z 549.53,A -85,B 0,C 180,E1 8703.107,E2 8703.107} C_VEL
LIN {X 0,Y 435.404,Z 549.53,A -85,B 0,C 180,E1 8709.874,E2 8709.874} C_VEL
LIN {X 0,Y 435.571,Z 549.53,A -85,B 0,C 180,E1 8716.74,E2 8716.74} C_VEL
LIN {X 0,Y 435.804,Z 549.53,A -85,B 0,C 180,E1 8722.013,E2 8722.013} C_VEL
LIN {X 0,Y 436.072,Z 549.53,A -85,B 0,C 180,E1 8728.011,E2 8728.011} C_VEL
LIN {X 0,Y 435.893,Z 549.53,A -85,B 0,C 180,E1 8733.984,E2 8733.984} C_VEL
LIN {X 0,Y 435.68,Z 549.53,A -85,B 0,C 180,E1 8740.007,E2 8740.007} C_VEL
LIN {X 0,Y 435.519,Z 549.53,A -85,B 0,C 180,E1 8746.149,E2 8746.149} C_VEL
LIN {X 0,Y 435.35,Z 549.53,A -85,B 0,C 180,E1 8752.493,E2 8752.493} C_VEL
LIN {X 0,Y 435.077,Z 549.53,A -85,B 0,C 180,E1 8759.158,E2 8759.158} C_VEL
LIN {X 0,Y 435.066,Z 549.879,A -85,B 0,C 180,E1 8763.996,E2 8763.996} C_VEL
LIN {X 0,Y 450.909,Z 587.497,A -85,B 0,C 180,E1 8767.338,E2 8767.338} C_VEL
LIN {X 0,Y 457.862,Z 610.546,A -85,B 0,C 180,E1 8769.447,E2 8769.447} C_VEL
LIN {X 0,Y 453.198,Z 647.027,A -85,B 0,C 180,E1 8772.14,E2 8772.14} C_VEL
LIN {X 0,Y 448.46,Z 679.247,A -85,B 0,C 180,E1 8775.419,E2 8775.419} C_VEL
LIN {X 0,Y 444.034,Z 707.7,A -85,B 0,C 180,E1 8779.313,E2 8779.313} C_VEL
LIN {X 0,Y 440.603,Z 730.829,A -85,B 0,C 180,E1 8783.539,E2 8783.539} C_VEL
LIN {X 0,Y 438.118,Z 750.418,A -85,B 0,C 180,E1 8788.432,E2 8788.432} C_VEL
LIN {X 0,Y 436.726,Z 765.267,A -85,B 0,C 180,E1 8793.837,E2 8793.837} C_VEL
LIN {X 0,Y 436.186,Z 773.55,A -85,B 0,C 180,E1 8798.622,E2 8798.622} C_VEL
LIN {X 0,Y 435.902,Z 777.374,A -85,B 0,C 180,E1 8803.863,E2 8803.863} C_VEL
LIN {X 0,Y 435.993,Z 776.577,A -85,B 0,C 180,E1 8807.97,E2 8807.97} C_VEL
LIN {X 0,Y 436.425,Z 771.073,A -85,B 0,C 180,E1 8813.022,E2 8813.022} C_VEL
LIN {X 0,Y 437.086,Z 760.617,A -85,B 0,C 180,E1 8818.011,E2 8818.011} C_VEL
LIN {X 0,Y 438.713,Z 745.371,A -85,B 0,C 180,E1 8822.963,E2 8822.963} C_VEL
LIN {X 0,Y 441.525,Z 725.026,A -85,B 0,C 180,E1 8827.632,E2 8827.632} C_VEL
LIN {X 0,Y 445.312,Z 700.474,A -85,B 0,C 180,E1 8831.766,E2 8831.766} C_VEL
LIN {X 0,Y 449.685,Z 671.723,A -85,B 0,C 180,E1 8835.371,E2 8835.371} C_VEL
LIN {X 0,Y 454.268,Z 638.342,A -85,B 0,C 180,E1 8838.455,E2 8838.455} C_VEL
LIN {X 0,Y 457.393,Z 607.021,A -85,B 0,C 180,E1 8840.598,E2 8840.598} C_VEL
LIN {X 0,Y 442.955,Z 567.133,A -85,B 0,C 180,E1 8844.126,E2 8844.126} C_VEL
LIN {X 0,Y 435.287,Z 549.53,A -85,B 0,C 180,E1 8845.753,E2 8845.753} C_VEL
LIN {X 0,Y 435.031,Z 549.53,A -85,B 0,C 180,E1 8851.464,E2 8851.464} C_VEL
LIN {X 0,Y 434.928,Z 549.53,A -85,B 0,C 180,E1 8858.794,E2 8858.794} C_VEL
LIN {X 0,Y 434.985,Z 549.53,A -85,B 0,C 180,E1 8864.111,E2 8864.111} C_VEL
LIN {X 0,Y 434.97,Z 550.234,A -85,B 0,C 180,E1 8867.968,E2 8867.968} C_VEL
LIN {X 0,Y 451.274,Z 584.93,A -85,B 0,C 180,E1 8870.406,E2 8870.406} C_VEL
LIN {X 0,Y 461.271,Z 608.263,A -85,B 0,C 180,E1 8871.814,E2 8871.814} C_VEL
LIN {X 0,Y 459.233,Z 638.674,A -85,B 0,C 180,E1 8872.74,E2 8872.74} C_VEL
LIN {X 0,Y 454.356,Z 655.204,A -85,B 0,C 180,E1 8873.169,E2 8873.169} C_VEL
LIN {X 0,Y 449.63,Z 669.351,A -85,B 0,C 180,E1 8873.641,E2 8873.641} C_VEL
LIN {X 0,Y 449.392,Z 671.321,A -85,B 0,C 180,E1 8873.748,E2 8873.748} C_VEL
LIN {X 0,Y 445.111,Z 709.491,A -85,B 0,C 180,E1 8876.227,E2 8876.227} C_VEL
LIN {X 0,Y 440.653,Z 745.013,A -85,B 0,C 180,E1 8879.415,E2 8879.415} C_VEL
LIN {X 0,Y 436.546,Z 776.394,A -85,B 0,C 180,E1 8883.199,E2 8883.199} C_VEL
LIN {X 0,Y 432.937,Z 804.141,A -85,B 0,C 180,E1 8887.68,E2 8887.68} C_VEL
LIN {X 0,Y 430.43,Z 826.424,A -85,B 0,C 180,E1 8892.602,E2 8892.602} C_VEL
LIN {X 0,Y 429.081,Z 841.383,A -85,B 0,C 180,E1 8897.258,E2 8897.258} C_VEL
LIN {X 0,Y 428.542,Z 851.165,A -85,B 0,C 180,E1 8901.875,E2 8901.875} C_VEL
LIN {X 0,Y 428.303,Z 855.894,A -85,B 0,C 180,E1 8905.945,E2 8905.945} C_VEL
LIN {X 0,Y 428.37,Z 857.5,A -85,B 0,C 180,E1 8909.999,E2 8909.999} C_VEL
LIN {X 0,Y 428.323,Z 855.899,A -85,B 0,C 180,E1 8914.053,E2 8914.053} C_VEL
LIN {X 0,Y 428.698,Z 849.396,A -85,B 0,C 180,E1 8919.191,E2 8919.191} C_VEL
LIN {X 0,Y 429.558,Z 837.183,A -85,B 0,C 180,E1 8924.283,E2 8924.283} C_VEL
LIN {X 0,Y 431.296,Z 818.92,A -85,B 0,C 180,E1 8929.374,E2 8929.374} C_VEL
LIN {X 0,Y 434.388,Z 795.052,A -85,B 0,C 180,E1 8934.176,E2 8934.176} C_VEL
LIN {X 0,Y 438.428,Z 767.039,A -85,B 0,C 180,E1 8938.39,E2 8938.39} C_VEL
LIN {X 0,Y 443.154,Z 735.038,A -85,B 0,C 180,E1 8942.019,E2 8942.019} C_VEL
LIN {X 0,Y 447.975,Z 700.846,A -85,B 0,C 180,E1 8944.905,E2 8944.905} C_VEL
LIN {X 0,Y 452.389,Z 664.036,A -85,B 0,C 180,E1 8947.146,E2 8947.146} C_VEL
LIN {X 0,Y 455.837,Z 625.552,A -85,B 0,C 180,E1 8948.708,E2 8948.708} C_VEL
LIN {X 0,Y 456.206,Z 609.214,A -85,B 0,C 180,E1 8949.222,E2 8949.222} C_VEL
LIN {X 0,Y 431.863,Z 559.856,A -85,B 0,C 180,E1 8952.777,E2 8952.777} C_VEL
LIN {X 0,Y 427.183,Z 550.828,A -85,B 0,C 180,E1 8953.493,E2 8953.493} C_VEL
LIN {X 0,Y 427.084,Z 549.53,A -85,B 0,C 180,E1 8953.71,E2 8953.71} C_VEL
LIN {X 0,Y 426.95,Z 549.53,A -85,B 0,C 180,E1 8960.34,E2 8960.34} C_VEL
LIN {X 0,Y 427.027,Z 549.53,A -85,B 0,C 180,E1 8965.444,E2 8965.444} C_VEL
LIN {X 0,Y 427.172,Z 549.53,A -85,B 0,C 180,E1 8970.256,E2 8970.256} C_VEL
LIN {X 0,Y 427.305,Z 549.53,A -85,B 0,C 180,E1 8977.108,E2 8977.108} C_VEL
LIN {X 0,Y 427.537,Z 549.53,A -85,B 0,C 180,E1 8983.547,E2 8983.547} C_VEL
LIN {X 0,Y 427.777,Z 549.53,A -85,B 0,C 180,E1 8989.811,E2 8989.811} C_VEL
LIN {X 0,Y 428.022,Z 549.53,A -85,B 0,C 180,E1 8995.947,E2 8995.947} C_VEL
LIN {X 0,Y 428.253,Z 549.53,A -85,B 0,C 180,E1 9002.03,E2 9002.03} C_VEL
LIN {X 0,Y 427.887,Z 549.53,A -85,B 0,C 180,E1 9008.141,E2 9008.141} C_VEL
LIN {X 0,Y 427.602,Z 549.53,A -85,B 0,C 180,E1 9014.355,E2 9014.355} C_VEL
LIN {X 0,Y 427.409,Z 549.53,A -85,B 0,C 180,E1 9020.751,E2 9020.751} C_VEL
LIN {X 0,Y 427.188,Z 549.53,A -85,B 0,C 180,E1 9027.619,E2 9027.619} C_VEL
LIN {X 0,Y 427.072,Z 549.53,A -85,B 0,C 180,E1 9032.13,E2 9032.13} C_VEL
LIN {X 0,Y 427.015,Z 549.53,A -85,B 0,C 180,E1 9038.736,E2 9038.736} C_VEL
LIN {X 0,Y 426.978,Z 549.53,A -85,B 0,C 180,E1 9045.174,E2 9045.174} C_VEL
LIN {X 0,Y 426.959,Z 549.53,A -85,B 0,C 180,E1 9051.28,E2 9051.28} C_VEL
LIN {X 0,Y 427.165,Z 549.53,A -85,B 0,C 180,E1 9058.29,E2 9058.29} C_VEL
LIN {X 0,Y 427.264,Z 549.53,A -85,B 0,C 180,E1 9064.835,E2 9064.835} C_VEL
LIN {X 0,Y 427.486,Z 549.53,A -85,B 0,C 180,E1 9071.413,E2 9071.413} C_VEL
LIN {X 0,Y 427.689,Z 549.53,A -85,B 0,C 180,E1 9077.738,E2 9077.738} C_VEL
LIN {X 0,Y 427.927,Z 549.53,A -85,B 0,C 180,E1 9083.908,E2 9083.908} C_VEL
LIN {X 0,Y 428.253,Z 549.53,A -85,B 0,C 180,E1 9090.001,E2 9090.001} C_VEL
LIN {X 0,Y 427.986,Z 549.53,A -85,B 0,C 180,E1 9096.093,E2 9096.093} C_VEL
LIN {X 0,Y 427.678,Z 549.53,A -85,B 0,C 180,E1 9102.265,E2 9102.265} C_VEL
LIN {X 0,Y 427.509,Z 549.53,A -85,B 0,C 180,E1 9108.588,E2 9108.588} C_VEL
LIN {X 0,Y 427.352,Z 549.53,A -85,B 0,C 180,E1 9115.161,E2 9115.161} C_VEL
LIN {X 0,Y 427.104,Z 549.53,A -85,B 0,C 180,E1 9122.124,E2 9122.124} C_VEL
LIN {X 0,Y 427.141,Z 549.694,A -85,B 0,C 180,E1 9123.162,E2 9123.162} C_VEL
LIN {X 0,Y 443.474,Z 588.276,A -85,B 0,C 180,E1 9126.69,E2 9126.69} C_VEL
LIN {X 0,Y 451.135,Z 611.912,A -85,B 0,C 180,E1 9128.959,E2 9128.959} C_VEL
LIN {X 0,Y 446.215,Z 648.422,A -85,B 0,C 180,E1 9131.709,E2 9131.709} C_VEL
LIN {X 0,Y 441.143,Z 681.098,A -85,B 0,C 180,E1 9135.108,E2 9135.108} C_VEL
LIN {X 0,Y 436.501,Z 709.51,A -85,B 0,C 180,E1 9139.1,E2 9139.1} C_VEL
LIN {X 0,Y 432.806,Z 733.185,A -85,B 0,C 180,E1 9143.573,E2 9143.573} C_VEL
LIN {X 0,Y 430.452,Z 751.002,A -85,B 0,C 180,E1 9148.152,E2 9148.152} C_VEL
LIN {X 0,Y 428.993,Z 764.932,A -85,B 0,C 180,E1 9153.28,E2 9153.28} C_VEL
LIN {X 0,Y 428.336,Z 773.244,A -85,B 0,C 180,E1 9158.21,E2 9158.21} C_VEL
LIN {X 0,Y 427.973,Z 777.303,A -85,B 0,C 180,E1 9163.555,E2 9163.555} C_VEL
LIN {X 0,Y 428.088,Z 776.741,A -85,B 0,C 180,E1 9167.744,E2 9167.744} C_VEL
LIN {X 0,Y 428.545,Z 771.683,A -85,B 0,C 180,E1 9172.893,E2 9172.893} C_VEL
LIN {X 0,Y 429.297,Z 762.009,A -85,B 0,C 180,E1 9177.975,E2 9177.975} C_VEL
LIN {X 0,Y 430.984,Z 747.022,A -85,B 0,C 180,E1 9183.016,E2 9183.016} C_VEL
LIN {X 0,Y 433.905,Z 726.941,A -85,B 0,C 180,E1 9187.767,E2 9187.767} C_VEL
LIN {X 0,Y 437.818,Z 702.678,A -85,B 0,C 180,E1 9191.971,E2 9191.971} C_VEL
LIN {X 0,Y 442.397,Z 674.294,A -85,B 0,C 180,E1 9195.631,E2 9195.631} C_VEL
LIN {X 0,Y 447.149,Z 641.487,A -85,B 0,C 180,E1 9198.758,E2 9198.758} C_VEL
LIN {X 0,Y 450.516,Z 609.582,A -85,B 0,C 180,E1 9201.022,E2 9201.022} C_VEL
LIN {X 0,Y 436.261,Z 569.208,A -85,B 0,C 180,E1 9204.743,E2 9204.743} C_VEL
LIN {X 0,Y 427.315,Z 549.53,A -85,B 0,C 180,E1 9206.717,E2 9206.717} C_VEL
LIN {X 0,Y 427.084,Z 549.53,A -85,B 0,C 180,E1 9212.119,E2 9212.119} C_VEL
LIN {X 0,Y 427.031,Z 549.53,A -85,B 0,C 180,E1 9218.736,E2 9218.736} C_VEL
LIN {X 0,Y 427.03,Z 549.53,A -85,B 0,C 180,E1 9225.155,E2 9225.155} C_VEL
LIN {X 0,Y 427.003,Z 549.53,A -85,B 0,C 180,E1 9226.988,E2 9226.988} C_VEL
LIN {X 0,Y 429.57,Z 555.339,A -85,B 0,C 180,E1 9227.47,E2 9227.47} C_VEL
LIN {X 0,Y 443.887,Z 585.206,A -85,B 0,C 180,E1 9229.732,E2 9229.732} C_VEL
LIN {X 0,Y 454.421,Z 611.367,A -85,B 0,C 180,E1 9231.363,E2 9231.363} C_VEL
LIN {X 0,Y 450.994,Z 654.925,A -85,B 0,C 180,E1 9232.922,E2 9232.922} C_VEL
LIN {X 0,Y 449.392,Z 671.321,A -85,B 0,C 180,E1 9233.748,E2 9233.748} C_VEL
LIN {X 0,Y 446.059,Z 683.407,A -85,B 0,C 180,E1 9234.303,E2 9234.303} C_VEL
LIN {X 0,Y 439.132,Z 700.686,A -85,B 0,C 180,E1 9235.14,E2 9235.14} C_VEL
LIN {X 0,Y 438.784,Z 702.596,A -85,B 0,C 180,E1 9235.271,E2 9235.271} C_VEL
LIN {X 0,Y 434.037,Z 739.135,A -85,B 0,C 180,E1 9238.449,E2 9238.449} C_VEL
LIN {X 0,Y 429.628,Z 770.785,A -85,B 0,C 180,E1 9242.146,E2 9242.146} C_VEL
LIN {X 0,Y 425.932,Z 798.288,A -85,B 0,C 180,E1 9246.427,E2 9246.427} C_VEL
LIN {X 0,Y 423.202,Z 821.151,A -85,B 0,C 180,E1 9251.216,E2 9251.216} C_VEL
LIN {X 0,Y 421.446,Z 838.361,A -85,B 0,C 180,E1 9256.255,E2 9256.255} C_VEL
LIN {X 0,Y 420.81,Z 848.647,A -85,B 0,C 180,E1 9260.681,E2 9260.681} C_VEL
LIN {X 0,Y 420.417,Z 855.479,A -85,B 0,C 180,E1 9265.869,E2 9265.869} C_VEL
LIN {X 0,Y 420.494,Z 857.208,A -85,B 0,C 180,E1 9269.999,E2 9269.999} C_VEL
LIN {X 0,Y 420.436,Z 854.589,A -85,B 0,C 180,E1 9275.164,E2 9275.164} C_VEL
LIN {X 0,Y 420.892,Z 846.723,A -85,B 0,C 180,E1 9280.361,E2 9280.361} C_VEL
LIN {X 0,Y 421.941,Z 833.152,A -85,B 0,C 180,E1 9285.611,E2 9285.611} C_VEL
LIN {X 0,Y 424.013,Z 814.18,A -85,B 0,C 180,E1 9290.646,E2 9290.646} C_VEL
LIN {X 0,Y 427.515,Z 789.413,A -85,B 0,C 180,E1 9295.449,E2 9295.449} C_VEL
LIN {X 0,Y 432.218,Z 759.236,A -85,B 0,C 180,E1 9299.788,E2 9299.788} C_VEL
LIN {X 0,Y 437.315,Z 726.119,A -85,B 0,C 180,E1 9303.34,E2 9303.34} C_VEL
LIN {X 0,Y 442.48,Z 690.478,A -85,B 0,C 180,E1 9306.147,E2 9306.147} C_VEL
LIN {X 0,Y 446.948,Z 652.54,A -85,B 0,C 180,E1 9308.247,E2 9308.247} C_VEL
LIN {X 0,Y 449.695,Z 612.086,A -85,B 0,C 180,E1 9309.723,E2 9309.723} C_VEL
LIN {X 0,Y 428.776,Z 568.851,A -85,B 0,C 180,E1 9312.89,E2 9312.89} C_VEL
LIN {X 0,Y 419.177,Z 550.27,A -85,B 0,C 180,E1 9314.399,E2 9314.399} C_VEL
LIN {X 0,Y 418.991,Z 549.53,A -85,B 0,C 180,E1 9319.432,E2 9319.432} C_VEL
LIN {X 0,Y 419.093,Z 549.53,A -85,B 0,C 180,E1 9326.192,E2 9326.192} C_VEL
LIN {X 0,Y 419.255,Z 549.53,A -85,B 0,C 180,E1 9332.006,E2 9332.006} C_VEL
LIN {X 0,Y 419.436,Z 549.53,A -85,B 0,C 180,E1 9338.845,E2 9338.845} C_VEL
LIN {X 0,Y 419.682,Z 549.53,A -85,B 0,C 180,E1 9345.377,E2 9345.377} C_VEL
LIN {X 0,Y 419.947,Z 549.53,A -85,B 0,C 180,E1 9351.713,E2 9351.713} C_VEL
LIN {X 0,Y 420.179,Z 549.53,A -85,B 0,C 180,E1 9357.939,E2 9357.939} C_VEL
LIN {X 0,Y 420.079,Z 549.53,A -85,B 0,C 180,E1 9364.138,E2 9364.138} C_VEL
LIN {X 0,Y 419.801,Z 549.53,A -85,B 0,C 180,E1 9370.393,E2 9370.393} C_VEL
LIN {X 0,Y 419.634,Z 549.53,A -85,B 0,C 180,E1 9376.781,E2 9376.781} C_VEL
LIN {X 0,Y 419.39,Z 549.53,A -85,B 0,C 180,E1 9383.402,E2 9383.402} C_VEL
LIN {X 0,Y 419.189,Z 549.53,A -85,B 0,C 180,E1 9390.38,E2 9390.38} C_VEL
LIN {X 0,Y 419.071,Z 549.53,A -85,B 0,C 180,E1 9397.898,E2 9397.898} C_VEL
LIN {X 0,Y 418.991,Z 549.53,A -85,B 0,C 180,E1 9403.722,E2 9403.722} C_VEL
LIN {X 0,Y 418.959,Z 549.53,A -85,B 0,C 180,E1 9409.422,E2 9409.422} C_VEL
LIN {X 0,Y 419.088,Z 549.53,A -85,B 0,C 180,E1 9416.2,E2 9416.2} C_VEL
LIN {X 0,Y 419.231,Z 549.53,A -85,B 0,C 180,E1 9421.999,E2 9421.999} C_VEL
LIN {X 0,Y 419.431,Z 549.53,A -85,B 0,C 180,E1 9428.841,E2 9428.841} C_VEL
LIN {X 0,Y 419.714,Z 549.53,A -85,B 0,C 180,E1 9435.374,E2 9435.374} C_VEL
LIN {X 0,Y 419.974,Z 549.53,A -85,B 0,C 180,E1 9441.71,E2 9441.71} C_VEL
LIN {X 0,Y 420.261,Z 549.53,A -85,B 0,C 180,E1 9447.936,E2 9447.936} C_VEL
LIN {X 0,Y 420.082,Z 549.53,A -85,B 0,C 180,E1 9454.135,E2 9454.135} C_VEL
LIN {X 0,Y 419.823,Z 549.53,A -85,B 0,C 180,E1 9460.389,E2 9460.389} C_VEL
LIN {X 0,Y 419.656,Z 549.53,A -85,B 0,C 180,E1 9466.777,E2 9466.777} C_VEL
LIN {X 0,Y 419.435,Z 549.53,A -85,B 0,C 180,E1 9473.396,E2 9473.396} C_VEL
LIN {X 0,Y 419.217,Z 549.53,A -85,B 0,C 180,E1 9480.374,E2 9480.374} C_VEL
LIN {X 0,Y 419.22,Z 549.78,A -85,B 0,C 180,E1 9482.296,E2 9482.296} C_VEL
LIN {X 0,Y 436.094,Z 589.063,A -85,B 0,C 180,E1 9486.02,E2 9486.02} C_VEL
LIN {X 0,Y 444.266,Z 613.904,A -85,B 0,C 180,E1 9488.494,E2 9488.494} C_VEL
LIN {X 0,Y 439.307,Z 649.439,A -85,B 0,C 180,E1 9491.227,E2 9491.227} C_VEL
LIN {X 0,Y 434.274,Z 680.699,A -85,B 0,C 180,E1 9494.512,E2 9494.512} C_VEL
LIN {X 0,Y 429.572,Z 707.795,A -85,B 0,C 180,E1 9498.294,E2 9498.294} C_VEL
LIN {X 0,Y 425.572,Z 731.825,A -85,B 0,C 180,E1 9502.781,E2 9502.781} C_VEL
LIN {X 0,Y 422.89,Z 750.472,A -85,B 0,C 180,E1 9507.513,E2 9507.513} C_VEL
LIN {X 0,Y 421.313,Z 764.67,A -85,B 0,C 180,E1 9512.656,E2 9512.656} C_VEL
LIN {X 0,Y 420.514,Z 773.565,A -85,B 0,C 180,E1 9517.783,E2 9517.783} C_VEL
LIN {X 0,Y 420.092,Z 777.809,A -85,B 0,C 180,E1 9523.238,E2 9523.238} C_VEL
LIN {X 0,Y 420.203,Z 777.525,A -85,B 0,C 180,E1 9527.511,E2 9527.511} C_VEL
LIN {X 0,Y 420.71,Z 772.799,A -85,B 0,C 180,E1 9532.781,E2 9532.781} C_VEL
LIN {X 0,Y 421.476,Z 763.407,A -85,B 0,C 180,E1 9537.937,E2 9537.937} C_VEL
LIN {X 0,Y 423.247,Z 748.675,A -85,B 0,C 180,E1 9543.072,E2 9543.072} C_VEL
LIN {X 0,Y 426.289,Z 728.86,A -85,B 0,C 180,E1 9547.906,E2 9547.906} C_VEL
LIN {X 0,Y 430.345,Z 704.903,A -85,B 0,C 180,E1 9552.182,E2 9552.182} C_VEL
LIN {X 0,Y 435.272,Z 675.826,A -85,B 0,C 180,E1 9556.023,E2 9556.023} C_VEL
LIN {X 0,Y 439.992,Z 644.691,A -85,B 0,C 180,E1 9559.076,E2 9559.076} C_VEL
LIN {X 0,Y 443.734,Z 612.28,A -85,B 0,C 180,E1 9561.45,E2 9561.45} C_VEL
LIN {X 0,Y 430.078,Z 572.64,A -85,B 0,C 180,E1 9565.278,E2 9565.278} C_VEL
LIN {X 0,Y 419.276,Z 549.53,A -85,B 0,C 180,E1 9567.762,E2 9567.762} C_VEL
LIN {X 0,Y 419.089,Z 549.53,A -85,B 0,C 180,E1 9575.306,E2 9575.306} C_VEL
LIN {X 0,Y 419.065,Z 549.53,A -85,B 0,C 180,E1 9580.647,E2 9580.647} C_VEL
LIN {X 0,Y 419.093,Z 549.76,A -85,B 0,C 180,E1 9585.927,E2 9585.927} C_VEL
LIN {X 0,Y 421.71,Z 555.426,A -85,B 0,C 180,E1 9586.469,E2 9586.469} C_VEL
LIN {X 0,Y 435.464,Z 582.867,A -85,B 0,C 180,E1 9588.834,E2 9588.834} C_VEL
LIN {X 0,Y 447.679,Z 613.131,A -85,B 0,C 180,E1 9590.862,E2 9590.862} C_VEL
LIN {X 0,Y 444.116,Z 654.848,A -85,B 0,C 180,E1 9592.419,E2 9592.419} C_VEL
LIN {X 0,Y 439.899,Z 693.589,A -85,B 0,C 180,E1 9594.638,E2 9594.638} C_VEL
LIN {X 0,Y 438.784,Z 702.596,A -85,B 0,C 180,E1 9595.271,E2 9595.271} C_VEL
LIN {X 0,Y 433.129,Z 717.547,A -85,B 0,C 180,E1 9596.235,E2 9596.235} C_VEL
LIN {X 0,Y 427.649,Z 731.944,A -85,B 0,C 180,E1 9597.344,E2 9597.344} C_VEL
LIN {X 0,Y 422.946,Z 764.944,A -85,B 0,C 180,E1 9601.066,E2 9601.066} C_VEL
LIN {X 0,Y 418.739,Z 794.141,A -85,B 0,C 180,E1 9605.471,E2 9605.471} C_VEL
LIN {X 0,Y 415.694,Z 817.827,A -85,B 0,C 180,E1 9610.31,E2 9610.31} C_VEL
LIN {X 0,Y 413.867,Z 835.019,A -85,B 0,C 180,E1 9615.161,E2 9615.161} C_VEL
LIN {X 0,Y 412.94,Z 847.78,A -85,B 0,C 180,E1 9620.502,E2 9620.502} C_VEL
LIN {X 0,Y 412.566,Z 854.704,A -85,B 0,C 180,E1 9625.79,E2 9625.79} C_VEL
LIN {X 0,Y 412.647,Z 856.47,A -85,B 0,C 180,E1 9629.999,E2 9629.999} C_VEL
LIN {X 0,Y 412.566,Z 853.865,A -85,B 0,C 180,E1 9635.263,E2 9635.263} C_VEL
LIN {X 0,Y 413.042,Z 845.981,A -85,B 0,C 180,E1 9640.56,E2 9640.56} C_VEL
LIN {X 0,Y 414.128,Z 832.363,A -85,B 0,C 180,E1 9645.914,E2 9645.914} C_VEL
LIN {X 0,Y 416.353,Z 813.328,A -85,B 0,C 180,E1 9651.044,E2 9651.044} C_VEL
LIN {X 0,Y 420.099,Z 788.591,A -85,B 0,C 180,E1 9655.911,E2 9655.911} C_VEL
LIN {X 0,Y 425.032,Z 757.844,A -85,B 0,C 180,E1 9660.385,E2 9660.385} C_VEL
LIN {X 0,Y 430.429,Z 724.883,A -85,B 0,C 180,E1 9663.945,E2 9663.945} C_VEL
LIN {X 0,Y 435.926,Z 687.72,A -85,B 0,C 180,E1 9666.871,E2 9666.871} C_VEL
LIN {X 0,Y 440.627,Z 650.096,A -85,B 0,C 180,E1 9668.926,E2 9668.926} C_VEL
LIN {X 0,Y 443.188,Z 614.81,A -85,B 0,C 180,E1 9670.244,E2 9670.244} C_VEL
LIN {X 0,Y 423.048,Z 572.888,A -85,B 0,C 180,E1 9673.412,E2 9673.412} C_VEL
LIN {X 0,Y 411.232,Z 549.932,A -85,B 0,C 180,E1 9675.331,E2 9675.331} C_VEL
LIN {X 0,Y 411.027,Z 549.53,A -85,B 0,C 180,E1 9681.236,E2 9681.236} C_VEL
LIN {X 0,Y 411.196,Z 549.53,A -85,B 0,C 180,E1 9687.872,E2 9687.872} C_VEL
LIN {X 0,Y 411.322,Z 549.53,A -85,B 0,C 180,E1 9693.792,E2 9693.792} C_VEL
LIN {X 0,Y 411.568,Z 549.53,A -85,B 0,C 180,E1 9700.67,E2 9700.67} C_VEL
LIN {X 0,Y 411.827,Z 549.53,A -85,B 0,C 180,E1 9707.261,E2 9707.261} C_VEL
LIN {X 0,Y 412.083,Z 549.53,A -85,B 0,C 180,E1 9713.676,E2 9713.676} C_VEL
LIN {X 0,Y 412.365,Z 549.53,A -85,B 0,C 180,E1 9720.004,E2 9720.004} C_VEL
LIN {X 0,Y 412.143,Z 549.53,A -85,B 0,C 180,E1 9726.332,E2 9726.332} C_VEL
LIN {X 0,Y 411.824,Z 549.53,A -85,B 0,C 180,E1 9732.748,E2 9732.748} C_VEL
LIN {X 0,Y 411.61,Z 549.53,A -85,B 0,C 180,E1 9739.337,E2 9739.337} C_VEL
LIN {X 0,Y 411.337,Z 549.53,A -85,B 0,C 180,E1 9746.217,E2 9746.217} C_VEL
LIN {X 0,Y 411.156,Z 549.53,A -85,B 0,C 180,E1 9753.534,E2 9753.534} C_VEL
LIN {X 0,Y 411.058,Z 549.53,A -85,B 0,C 180,E1 9759.332,E2 9759.332} C_VEL
LIN {X 0,Y 411.011,Z 549.53,A -85,B 0,C 180,E1 9765.581,E2 9765.581} C_VEL
LIN {X 0,Y 411.011,Z 549.53,A -85,B 0,C 180,E1 9771.228,E2 9771.228} C_VEL
LIN {X 0,Y 411.186,Z 549.53,A -85,B 0,C 180,E1 9777.882,E2 9777.882} C_VEL
LIN {X 0,Y 411.314,Z 549.53,A -85,B 0,C 180,E1 9783.787,E2 9783.787} C_VEL
LIN {X 0,Y 411.605,Z 549.53,A -85,B 0,C 180,E1 9790.668,E2 9790.668} C_VEL
LIN {X 0,Y 411.854,Z 549.53,A -85,B 0,C 180,E1 9797.258,E2 9797.258} C_VEL
LIN {X 0,Y 412.112,Z 549.53,A -85,B 0,C 180,E1 9803.673,E2 9803.673} C_VEL
LIN {X 0,Y 412.45,Z 549.53,A -85,B 0,C 180,E1 9810.001,E2 9810.001} C_VEL
LIN {X 0,Y 412.063,Z 549.53,A -85,B 0,C 180,E1 9817.195,E2 9817.195} C_VEL
LIN {X 0,Y 411.838,Z 549.53,A -85,B 0,C 180,E1 9822.744,E2 9822.744} C_VEL
LIN {X 0,Y 411.631,Z 549.53,A -85,B 0,C 180,E1 9829.333,E2 9829.333} C_VEL
LIN {X 0,Y 411.396,Z 549.53,A -85,B 0,C 180,E1 9836.209,E2 9836.209} C_VEL
LIN {X 0,Y 411.333,Z 549.726,A -85,B 0,C 180,E1 9841.411,E2 9841.411} C_VEL
LIN {X 0,Y 428.008,Z 588.116,A -85,B 0,C 180,E1 9845.151,E2 9845.151} C_VEL
LIN {X 0,Y 437.394,Z 617.079,A -85,B 0,C 180,E1 9848.114,E2 9848.114} C_VEL
LIN {X 0,Y 432.182,Z 652.016,A -85,B 0,C 180,E1 9850.881,E2 9850.881} C_VEL
LIN {X 0,Y 426.919,Z 683.009,A -85,B 0,C 180,E1 9854.235,E2 9854.235} C_VEL
LIN {X 0,Y 421.979,Z 710.256,A -85,B 0,C 180,E1 9858.167,E2 9858.167} C_VEL
LIN {X 0,Y 417.98,Z 732.925,A -85,B 0,C 180,E1 9862.518,E2 9862.518} C_VEL
LIN {X 0,Y 415.076,Z 752.116,A -85,B 0,C 180,E1 9867.538,E2 9867.538} C_VEL
LIN {X 0,Y 413.443,Z 765.972,A -85,B 0,C 180,E1 9872.753,E2 9872.753} C_VEL
LIN {X 0,Y 412.702,Z 774.037,A -85,B 0,C 180,E1 9877.47,E2 9877.47} C_VEL
LIN {X 0,Y 412.223,Z 778.45,A -85,B 0,C 180,E1 9882.908,E2 9882.908} C_VEL
LIN {X 0,Y 412.31,Z 778.394,A -85,B 0,C 180,E1 9887.267,E2 9887.267} C_VEL
LIN {X 0,Y 412.868,Z 773.653,A -85,B 0,C 180,E1 9892.857,E2 9892.857} C_VEL
LIN {X 0,Y 413.686,Z 764.799,A -85,B 0,C 180,E1 9897.898,E2 9897.898} C_VEL
LIN {X 0,Y 415.5,Z 750.335,A -85,B 0,C 180,E1 9903.129,E2 9903.129} C_VEL
LIN {X 0,Y 418.652,Z 730.787,A -85,B 0,C 180,E1 9908.051,E2 9908.051} C_VEL
LIN {X 0,Y 422.887,Z 707.136,A -85,B 0,C 180,E1 9912.4,E2 9912.4} C_VEL
LIN {X 0,Y 427.901,Z 678.543,A -85,B 0,C 180,E1 9916.306,E2 9916.306} C_VEL
LIN {X 0,Y 433.106,Z 646.562,A -85,B 0,C 180,E1 9919.523,E2 9919.523} C_VEL
LIN {X 0,Y 437.054,Z 615.236,A -85,B 0,C 180,E1 9921.88,E2 9921.88} C_VEL
LIN {X 0,Y 424.383,Z 577.102,A -85,B 0,C 180,E1 9925.721,E2 9925.721} C_VEL
LIN {X 0,Y 413.881,Z 555.348,A -85,B 0,C 180,E1 9928.244,E2 9928.244} C_VEL
LIN {X 0,Y 411.352,Z 550.435,A -85,B 0,C 180,E1 9928.873,E2 9928.873} C_VEL
LIN {X 0,Y 411.309,Z 549.53,A -85,B 0,C 180,E1 9929.051,E2 9929.051} C_VEL
LIN {X 0,Y 411.145,Z 549.53,A -85,B 0,C 180,E1 9936.094,E2 9936.094} C_VEL
LIN {X 0,Y 411.077,Z 549.53,A -85,B 0,C 180,E1 9942.553,E2 9942.553} C_VEL
LIN {X 0,Y 411.266,Z 550.12,A -85,B 0,C 180,E1 9944.722,E2 9944.722} C_VEL
LIN {X 0,Y 414.034,Z 555.55,A -85,B 0,C 180,E1 9945.365,E2 9945.365} C_VEL
LIN {X 0,Y 427.268,Z 581.074,A -85,B 0,C 180,E1 9947.889,E2 9947.889} C_VEL
LIN {X 0,Y 440.931,Z 615.116,A -85,B 0,C 180,E1 9950.353,E2 9950.353} C_VEL
LIN {X 0,Y 437.061,Z 656.931,A -85,B 0,C 180,E1 9952,E2 9952} C_VEL
LIN {X 0,Y 432.654,Z 694.965,A -85,B 0,C 180,E1 9954.268,E2 9954.268} C_VEL
LIN {X 0,Y 427.845,Z 730.321,A -85,B 0,C 180,E1 9957.187,E2 9957.187} C_VEL
LIN {X 0,Y 427.649,Z 731.944,A -85,B 0,C 180,E1 9957.344,E2 9957.344} C_VEL
LIN {X 0,Y 425.516,Z 739.001,A -85,B 0,C 180,E1 9957.982,E2 9957.982} C_VEL
LIN {X 0,Y 416.5,Z 757.4,A -85,B 0,C 180,E1 9959.751,E2 9959.751} C_VEL
LIN {X 0,Y 416.204,Z 758.989,A -85,B 0,C 180,E1 9959.952,E2 9959.952} C_VEL
LIN {X 0,Y 411.965,Z 787.243,A -85,B 0,C 180,E1 9964.053,E2 9964.053} C_VEL
LIN {X 0,Y 408.47,Z 811.856,A -85,B 0,C 180,E1 9968.813,E2 9968.813} C_VEL
LIN {X 0,Y 406.349,Z 830.641,A -85,B 0,C 180,E1 9973.772,E2 9973.772} C_VEL
LIN {X 0,Y 405.197,Z 844.816,A -85,B 0,C 180,E1 9979.231,E2 9979.231} C_VEL
LIN {X 0,Y 404.794,Z 851.773,A -85,B 0,C 180,E1 9983.556,E2 9983.556} C_VEL
LIN {X 0,Y 404.721,Z 855.248,A -85,B 0,C 180,E1 9987.855,E2 9987.855} C_VEL
LIN {X 0,Y 404.779,Z 855.315,A -85,B 0,C 180,E1 9992.143,E2 9992.143} C_VEL
LIN {X 0,Y 404.812,Z 851.975,A -85,B 0,C 180,E1 9996.442,E2 9996.442} C_VEL
LIN {X 0,Y 405.294,Z 842.97,A -85,B 0,C 180,E1 10001.856,E2 10001.856} C_VEL
LIN {X 0,Y 406.553,Z 829.898,A -85,B 0,C 180,E1 10006.775,E2 10006.775} C_VEL
LIN {X 0,Y 409.157,Z 809.77,A -85,B 0,C 180,E1 10012.072,E2 10012.072} C_VEL
LIN {X 0,Y 413.206,Z 784.311,A -85,B 0,C 180,E1 10016.964,E2 10016.964} C_VEL
LIN {X 0,Y 418.147,Z 755.487,A -85,B 0,C 180,E1 10021.115,E2 10021.115} C_VEL
LIN {X 0,Y 423.657,Z 722.964,A -85,B 0,C 180,E1 10024.626,E2 10024.626} C_VEL
LIN {X 0,Y 429.39,Z 686.156,A -85,B 0,C 180,E1 10027.528,E2 10027.528} C_VEL
LIN {X 0,Y 434.443,Z 646.897,A -85,B 0,C 180,E1 10029.659,E2 10029.659} C_VEL
LIN {X 0,Y 436.621,Z 617.35,A -85,B 0,C 180,E1 10030.794,E2 10030.794} C_VEL
LIN {X 0,Y 416.593,Z 575.313,A -85,B 0,C 180,E1 10034.069,E2 10034.069} C_VEL
LIN {X 0,Y 403.252,Z 550.5,A -85,B 0,C 180,E1 10036.273,E2 10036.273} C_VEL
LIN {X 0,Y 403.154,Z 549.53,A -85,B 0,C 180,E1 10036.42,E2 10036.42} C_VEL
LIN {X 0,Y 403.107,Z 549.53,A -85,B 0,C 180,E1 10043.068,E2 10043.068} C_VEL
LIN {X 0,Y 403.282,Z 549.53,A -85,B 0,C 180,E1 10049.71,E2 10049.71} C_VEL
LIN {X 0,Y 403.421,Z 549.53,A -85,B 0,C 180,E1 10055.622,E2 10055.622} C_VEL
LIN {X 0,Y 403.726,Z 549.53,A -85,B 0,C 180,E1 10062.547,E2 10062.547} C_VEL
LIN {X 0,Y 403.971,Z 549.53,A -85,B 0,C 180,E1 10069.204,E2 10069.204} C_VEL
LIN {X 0,Y 404.28,Z 549.53,A -85,B 0,C 180,E1 10075.709,E2 10075.709} C_VEL
LIN {X 0,Y 404.529,Z 549.53,A -85,B 0,C 180,E1 10082.149,E2 10082.149} C_VEL
LIN {X 0,Y 404.103,Z 549.53,A -85,B 0,C 180,E1 10088.624,E2 10088.624} C_VEL
LIN {X 0,Y 403.809,Z 549.53,A -85,B 0,C 180,E1 10095.22,E2 10095.22} C_VEL
LIN {X 0,Y 403.57,Z 549.53,A -85,B 0,C 180,E1 10102.039,E2 10102.039} C_VEL
LIN {X 0,Y 403.308,Z 549.53,A -85,B 0,C 180,E1 10109.216,E2 10109.216} C_VEL
LIN {X 0,Y 403.182,Z 549.53,A -85,B 0,C 180,E1 10114.295,E2 10114.295} C_VEL
LIN {X 0,Y 403.111,Z 549.53,A -85,B 0,C 180,E1 10121.308,E2 10121.308} C_VEL
LIN {X 0,Y 403.083,Z 549.53,A -85,B 0,C 180,E1 10127.46,E2 10127.46} C_VEL
LIN {X 0,Y 403.09,Z 549.53,A -85,B 0,C 180,E1 10133.061,E2 10133.061} C_VEL
LIN {X 0,Y 403.274,Z 549.53,A -85,B 0,C 180,E1 10139.72,E2 10139.72} C_VEL
LIN {X 0,Y 403.426,Z 549.53,A -85,B 0,C 180,E1 10145.618,E2 10145.618} C_VEL
LIN {X 0,Y 403.76,Z 549.53,A -85,B 0,C 180,E1 10152.544,E2 10152.544} C_VEL
LIN {X 0,Y 403.998,Z 549.53,A -85,B 0,C 180,E1 10159.201,E2 10159.201} C_VEL
LIN {X 0,Y 404.381,Z 549.53,A -85,B 0,C 180,E1 10165.706,E2 10165.706} C_VEL
LIN {X 0,Y 404.534,Z 549.53,A -85,B 0,C 180,E1 10172.146,E2 10172.146} C_VEL
LIN {X 0,Y 404.122,Z 549.53,A -85,B 0,C 180,E1 10178.62,E2 10178.62} C_VEL
LIN {X 0,Y 403.829,Z 549.53,A -85,B 0,C 180,E1 10185.216,E2 10185.216} C_VEL
LIN {X 0,Y 403.617,Z 549.53,A -85,B 0,C 180,E1 10192.033,E2 10192.033} C_VEL
LIN {X 0,Y 403.368,Z 549.53,A -85,B 0,C 180,E1 10199.208,E2 10199.208} C_VEL
LIN {X 0,Y 403.356,Z 549.53,A -85,B 0,C 180,E1 10200.462,E2 10200.462} C_VEL
LIN {X 0,Y 412.045,Z 568.887,A -85,B 0,C 180,E1 10202.364,E2 10202.364} C_VEL
LIN {X 0,Y 425.296,Z 601.95,A -85,B 0,C 180,E1 10205.788,E2 10205.788} C_VEL
LIN {X 0,Y 430.551,Z 619.572,A -85,B 0,C 180,E1 10207.668,E2 10207.668} C_VEL
LIN {X 0,Y 425.023,Z 654.695,A -85,B 0,C 180,E1 10210.536,E2 10210.536} C_VEL
LIN {X 0,Y 419.231,Z 686.983,A -85,B 0,C 180,E1 10214.161,E2 10214.161} C_VEL
LIN {X 0,Y 413.901,Z 715.37,A -85,B 0,C 180,E1 10218.491,E2 10218.491} C_VEL
LIN {X 0,Y 409.588,Z 738.749,A -85,B 0,C 180,E1 10223.344,E2 10223.344} C_VEL
LIN {X 0,Y 406.806,Z 756.873,A -85,B 0,C 180,E1 10228.593,E2 10228.593} C_VEL
LIN {X 0,Y 405.4,Z 768.969,A -85,B 0,C 180,E1 10233.683,E2 10233.683} C_VEL
LIN {X 0,Y 404.686,Z 776.856,A -85,B 0,C 180,E1 10239.285,E2 10239.285} C_VEL
LIN {X 0,Y 404.324,Z 779.565,A -85,B 0,C 180,E1 10244.799,E2 10244.799} C_VEL
LIN {X 0,Y 404.571,Z 778.142,A -85,B 0,C 180,E1 10249.211,E2 10249.211} C_VEL
LIN {X 0,Y 405.259,Z 772.103,A -85,B 0,C 180,E1 10254.636,E2 10254.636} C_VEL
LIN {X 0,Y 406.495,Z 761.138,A -85,B 0,C 180,E1 10259.996,E2 10259.996} C_VEL
LIN {X 0,Y 408.988,Z 744.575,A -85,B 0,C 180,E1 10265.306,E2 10265.306} C_VEL
LIN {X 0,Y 412.722,Z 723.863,A -85,B 0,C 180,E1 10270.03,E2 10270.03} C_VEL
LIN {X 0,Y 417.679,Z 697.624,A -85,B 0,C 180,E1 10274.426,E2 10274.426} C_VEL
LIN {X 0,Y 422.703,Z 669.728,A -85,B 0,C 180,E1 10277.916,E2 10277.916} C_VEL
LIN {X 0,Y 428.099,Z 636.556,A -85,B 0,C 180,E1 10280.978,E2 10280.978} C_VEL
LIN {X 0,Y 430.073,Z 617.164,A -85,B 0,C 180,E1 10282.444,E2 10282.444} C_VEL
LIN {X 0,Y 418.573,Z 580.908,A -85,B 0,C 180,E1 10286.249,E2 10286.249} C_VEL
LIN {X 0,Y 409.078,Z 560.819,A -85,B 0,C 180,E1 10288.755,E2 10288.755} C_VEL
LIN {X 0,Y 403.41,Z 550.652,A -85,B 0,C 180,E1 10290.317,E2 10290.317} C_VEL
LIN {X 0,Y 403.298,Z 549.53,A -85,B 0,C 180,E1 10290.585,E2 10290.585} C_VEL
LIN {X 0,Y 403.128,Z 549.53,A -85,B 0,C 180,E1 10296.929,E2 10296.929} C_VEL
LIN {X 0,Y 403.175,Z 549.571,A -85,B 0,C 180,E1 10303.189,E2 10303.189} C_VEL
LIN {X 0,Y 405.54,Z 555.105,A -85,B 0,C 180,E1 10303.904,E2 10303.904} C_VEL
LIN {X 0,Y 413.424,Z 568.361,A -85,B 0,C 180,E1 10305.71,E2 10305.71} C_VEL
LIN {X 0,Y 424.876,Z 592.735,A -85,B 0,C 180,E1 10307.961,E2 10307.961} C_VEL
LIN {X 0,Y 434.176,Z 618.691,A -85,B 0,C 180,E1 10309.875,E2 10309.875} C_VEL
LIN {X 0,Y 429.741,Z 661.757,A -85,B 0,C 180,E1 10311.693,E2 10311.693} C_VEL
LIN {X 0,Y 424.684,Z 701.837,A -85,B 0,C 180,E1 10314.281,E2 10314.281} C_VEL
LIN {X 0,Y 419.378,Z 738.518,A -85,B 0,C 180,E1 10317.593,E2 10317.593} C_VEL
LIN {X 0,Y 416.204,Z 758.989,A -85,B 0,C 180,E1 10319.952,E2 10319.952} C_VEL
LIN {X 0,Y 412.449,Z 768.521,A -85,B 0,C 180,E1 10321.105,E2 10321.105} C_VEL
LIN {X 0,Y 405.18,Z 781.854,A -85,B 0,C 180,E1 10322.884,E2 10322.884} C_VEL
LIN {X 0,Y 404.873,Z 783.295,A -85,B 0,C 180,E1 10323.114,E2 10323.114} C_VEL
LIN {X 0,Y 400.973,Z 809.434,A -85,B 0,C 180,E1 10328.106,E2 10328.106} C_VEL
LIN {X 0,Y 398.691,Z 827.816,A -85,B 0,C 180,E1 10332.883,E2 10332.883} C_VEL
LIN {X 0,Y 397.449,Z 841.562,A -85,B 0,C 180,E1 10337.905,E2 10337.905} C_VEL
LIN {X 0,Y 397.001,Z 849.826,A -85,B 0,C 180,E1 10342.51,E2 10342.51} C_VEL
LIN {X 0,Y 396.868,Z 854.493,A -85,B 0,C 180,E1 10347.813,E2 10347.813} C_VEL
LIN {X 0,Y 396.925,Z 854.584,A -85,B 0,C 180,E1 10352.185,E2 10352.185} C_VEL
LIN {X 0,Y 396.999,Z 850.175,A -85,B 0,C 180,E1 10357.487,E2 10357.487} C_VEL
LIN {X 0,Y 397.697,Z 839.787,A -85,B 0,C 180,E1 10363.203,E2 10363.203} C_VEL
LIN {X 0,Y 399.428,Z 823.54,A -85,B 0,C 180,E1 10368.795,E2 10368.795} C_VEL
LIN {X 0,Y 402.653,Z 801.965,A -85,B 0,C 180,E1 10374.024,E2 10374.024} C_VEL
LIN {X 0,Y 407.099,Z 776.468,A -85,B 0,C 180,E1 10378.609,E2 10378.609} C_VEL
LIN {X 0,Y 412.663,Z 745.886,A -85,B 0,C 180,E1 10382.732,E2 10382.732} C_VEL
LIN {X 0,Y 418.691,Z 711.722,A -85,B 0,C 180,E1 10386.148,E2 10386.148} C_VEL
LIN {X 0,Y 424.2,Z 675.474,A -85,B 0,C 180,E1 10388.779,E2 10388.779} C_VEL
LIN {X 0,Y 429.077,Z 636.178,A -85,B 0,C 180,E1 10390.702,E2 10390.702} C_VEL
LIN {X 0,Y 429.932,Z 619.722,A -85,B 0,C 180,E1 10391.343,E2 10391.343} C_VEL
LIN {X 0,Y 412.317,Z 582.092,A -85,B 0,C 180,E1 10394.372,E2 10394.372} C_VEL
LIN {X 0,Y 395.356,Z 550.888,A -85,B 0,C 180,E1 10397.253,E2 10397.253} C_VEL
LIN {X 0,Y 395.215,Z 549.53,A -85,B 0,C 180,E1 10397.461,E2 10397.461} C_VEL
LIN {X 0,Y 395.228,Z 549.53,A -85,B 0,C 180,E1 10404.933,E2 10404.933} C_VEL
LIN {X 0,Y 395.385,Z 549.53,A -85,B 0,C 180,E1 10411.731,E2 10411.731} C_VEL
LIN {X 0,Y 395.548,Z 549.53,A -85,B 0,C 180,E1 10417.5,E2 10417.5} C_VEL
LIN {X 0,Y 395.85,Z 549.53,A -85,B 0,C 180,E1 10424.475,E2 10424.475} C_VEL
LIN {X 0,Y 396.175,Z 549.53,A -85,B 0,C 180,E1 10431.212,E2 10431.212} C_VEL
LIN {X 0,Y 396.481,Z 549.53,A -85,B 0,C 180,E1 10437.816,E2 10437.816} C_VEL
LIN {X 0,Y 396.614,Z 549.53,A -85,B 0,C 180,E1 10442.192,E2 10442.192} C_VEL
LIN {X 0,Y 396.173,Z 549.53,A -85,B 0,C 180,E1 10448.798,E2 10448.798} C_VEL
LIN {X 0,Y 395.863,Z 549.53,A -85,B 0,C 180,E1 10455.534,E2 10455.534} C_VEL
LIN {X 0,Y 395.593,Z 549.53,A -85,B 0,C 180,E1 10462.507,E2 10462.507} C_VEL
LIN {X 0,Y 395.381,Z 549.53,A -85,B 0,C 180,E1 10469.86,E2 10469.86} C_VEL
LIN {X 0,Y 395.164,Z 549.53,A -85,B 0,C 180,E1 10476.429,E2 10476.429} C_VEL
LIN {X 0,Y 395.176,Z 549.53,A -85,B 0,C 180,E1 10483.286,E2 10483.286} C_VEL
LIN {X 0,Y 395.164,Z 549.53,A -85,B 0,C 180,E1 10490.028,E2 10490.028} C_VEL
LIN {X 0,Y 395.288,Z 549.53,A -85,B 0,C 180,E1 10497.573,E2 10497.573} C_VEL
